# B&R Automation Studio project testovaci_pneu_stan (part 4)

#### multiword_types.h
```c
/*
 * multiword_types.h
 *
 * Academic License - for use in teaching, academic research, and meeting
 * course requirements at degree granting institutions only.  Not for
 * government, commercial, or other organizational use.
 *
 * Code generation for model "reg_FF_PI_pl_regr_stiff".
 *
 * Model version              : 1.135
 * Simulink Coder version : 9.6 (R2021b) 14-May-2021
 * C source code generated on : Tue Sep 27 10:51:43 2022
 *
 * Target selection: bur_grt.tlc
 * Note: GRT includes extra infrastructure and instrumentation for prototyping
 * Embedded hardware selection: Intel->x86/Pentium
 * Code generation objectives: Unspecified
 * Validation result: Not run
 */

#ifndef MULTIWORD_TYPES_H
#define MULTIWORD_TYPES_H
#include "rtwtypes.h"

/*
 * MultiWord supporting definitions
 */
typedef long int long_T;

/*
 * MultiWord types
 */
typedef struct {
  uint32_T chunks[2];
} int64m_T;

typedef struct {
  int64m_T re;
  int64m_T im;
} cint64m_T;

typedef struct {
  uint32_T chunks[2];
} uint64m_T;

typedef struct {
  uint64m_T re;
  uint64m_T im;
} cuint64m_T;

typedef struct {
  uint32_T chunks[3];
} int96m_T;

typedef struct {
  int96m_T re;
  int96m_T im;
} cint96m_T;

typedef struct {
  uint32_T chunks[3];
} uint96m_T;

typedef struct {
  uint96m_T re;
  uint96m_T im;
} cuint96m_T;

typedef struct {
  uint32_T chunks[4];
} int128m_T;

typedef struct {
  int128m_T re;
  int128m_T im;
} cint128m_T;

typedef struct {
  uint32_T chunks[4];
} uint128m_T;

typedef struct {
  uint128m_T re;
  uint128m_T im;
} cuint128m_T;

typedef struct {
  uint32_T chunks[5];
} int160m_T;

typedef struct {
  int160m_T re;
  int160m_T im;
} cint160m_T;

typedef struct {
  uint32_T chunks[5];
} uint160m_T;

typedef struct {
  uint160m_T re;
  uint160m_T im;
} cuint160m_T;

typedef struct {
  uint32_T chunks[6];
} int192m_T;

typedef struct {
  int192m_T re;
  int192m_T im;
} cint192m_T;

typedef struct {
  uint32_T chunks[6];
} uint192m_T;

typedef struct {
  uint192m_T re;
  uint192m_T im;
} cuint192m_T;

typedef struct {
  uint32_T chunks[7];
} int224m_T;

typedef struct {
  int224m_T re;
  int224m_T im;
} cint224m_T;

typedef struct {
  uint32_T chunks[7];
} uint224m_T;

typedef struct {
  uint224m_T re;
  uint224m_T im;
} cuint224m_T;

typedef struct {
  uint32_T chunks[8];
} int256m_T;

typedef struct {
  int256m_T re;
  int256m_T im;
} cint256m_T;

typedef struct {
  uint32_T chunks[8];
} uint256m_T;

typedef struct {
  uint256m_T re;
  uint256m_T im;
} cuint256m_T;

typedef struct {
  uint32_T chunks[9];
} int288m_T;

typedef struct {
  int288m_T re;
  int288m_T im;
} cint288m_T;

typedef struct {
  uint32_T chunks[9];
} uint288m_T;

typedef struct {
  uint288m_T re;
  uint288m_T im;
} cuint288m_T;

typedef struct {
  uint32_T chunks[10];
} int320m_T;

typedef struct {
  int320m_T re;
  int320m_T im;
} cint320m_T;

typedef struct {
  uint32_T chunks[10];
} uint320m_T;

typedef struct {
  uint320m_T re;
  uint320m_T im;
} cuint320m_T;

typedef struct {
  uint32_T chunks[11];
} int352m_T;

typedef struct {
  int352m_T re;
  int352m_T im;
} cint352m_T;

typedef struct {
  uint32_T chunks[11];
} uint352m_T;

typedef struct {
  uint352m_T re;
  uint352m_T im;
} cuint352m_T;

typedef struct {
  uint32_T chunks[12];
} int384m_T;

typedef struct {
  int384m_T re;
  int384m_T im;
} cint384m_T;

typedef struct {
  uint32_T chunks[12];
} uint384m_T;

typedef struct {
  uint384m_T re;
  uint384m_T im;
} cuint384m_T;

typedef struct {
  uint32_T chunks[13];
} int416m_T;

typedef struct {
  int416m_T re;
  int416m_T im;
} cint416m_T;

typedef struct {
  uint32_T chunks[13];
} uint416m_T;

typedef struct {
  uint416m_T re;
  uint416m_T im;
} cuint416m_T;

typedef struct {
  uint32_T chunks[14];
} int448m_T;

typedef struct {
  int448m_T re;
  int448m_T im;
} cint448m_T;

typedef struct {
  uint32_T chunks[14];
} uint448m_T;

typedef struct {
  uint448m_T re;
  uint448m_T im;
} cuint448m_T;

typedef struct {
  uint32_T chunks[15];
} int480m_T;

typedef struct {
  int480m_T re;
  int480m_T im;
} cint480m_T;

typedef struct {
  uint32_T chunks[15];
} uint480m_T;

typedef struct {
  uint480m_T re;
  uint480m_T im;
} cuint480m_T;

typedef struct {
  uint32_T chunks[16];
} int512m_T;

typedef struct {
  int512m_T re;
  int512m_T im;
} cint512m_T;

typedef struct {
  uint32_T chunks[16];
} uint512m_T;

typedef struct {
  uint512m_T re;
  uint512m_T im;
} cuint512m_T;

typedef struct {
  uint32_T chunks[17];
} int544m_T;

typedef struct {
  int544m_T re;
  int544m_T im;
} cint544m_T;

typedef struct {
  uint32_T chunks[17];
} uint544m_T;

typedef struct {
  uint544m_T re;
  uint544m_T im;
} cuint544m_T;

typedef struct {
  uint32_T chunks[18];
} int576m_T;

typedef struct {
  int576m_T re;
  int576m_T im;
} cint576m_T;

typedef struct {
  uint32_T chunks[18];
} uint576m_T;

typedef struct {
  uint576m_T re;
  uint576m_T im;
} cuint576m_T;

typedef struct {
  uint32_T chunks[19];
} int608m_T;

typedef struct {
  int608m_T re;
  int608m_T im;
} cint608m_T;

typedef struct {
  uint32_T chunks[19];
} uint608m_T;

typedef struct {
  uint608m_T re;
  uint608m_T im;
} cuint608m_T;

typedef struct {
  uint32_T chunks[20];
} int640m_T;

typedef struct {
  int640m_T re;
  int640m_T im;
} cint640m_T;

typedef struct {
  uint32_T chunks[20];
} uint640m_T;

typedef struct {
  uint640m_T re;
  uint640m_T im;
} cuint640m_T;

typedef struct {
  uint32_T chunks[21];
} int672m_T;

typedef struct {
  int672m_T re;
  int672m_T im;
} cint672m_T;

typedef struct {
  uint32_T chunks[21];
} uint672m_T;

typedef struct {
  uint672m_T re;
  uint672m_T im;
} cuint672m_T;

typedef struct {
  uint32_T chunks[22];
} int704m_T;

typedef struct {
  int704m_T re;
  int704m_T im;
} cint704m_T;

typedef struct {
  uint32_T chunks[22];
} uint704m_T;

typedef struct {
  uint704m_T re;
  uint704m_T im;
} cuint704m_T;

typedef struct {
  uint32_T chunks[23];
} int736m_T;

typedef struct {
  int736m_T re;
  int736m_T im;
} cint736m_T;

typedef struct {
  uint32_T chunks[23];
} uint736m_T;

typedef struct {
  uint736m_T re;
  uint736m_T im;
} cuint736m_T;

typedef struct {
  uint32_T chunks[24];
} int768m_T;

typedef struct {
  int768m_T re;
  int768m_T im;
} cint768m_T;

typedef struct {
  uint32_T chunks[24];
} uint768m_T;

typedef struct {
  uint768m_T re;
  uint768m_T im;
} cuint768m_T;

typedef struct {
  uint32_T chunks[25];
} int800m_T;

typedef struct {
  int800m_T re;
  int800m_T im;
} cint800m_T;

typedef struct {
  uint32_T chunks[25];
} uint800m_T;

typedef struct {
  uint800m_T re;
  uint800m_T im;
} cuint800m_T;

typedef struct {
  uint32_T chunks[26];
} int832m_T;

typedef struct {
  int832m_T re;
  int832m_T im;
} cint832m_T;

typedef struct {
  uint32_T chunks[26];
} uint832m_T;

typedef struct {
  uint832m_T re;
  uint832m_T im;
} cuint832m_T;

typedef struct {
  uint32_T chunks[27];
} int864m_T;

typedef struct {
  int864m_T re;
  int864m_T im;
} cint864m_T;

typedef struct {
  uint32_T chunks[27];
} uint864m_T;

typedef struct {
  uint864m_T re;
  uint864m_T im;
} cuint864m_T;

typedef struct {
  uint32_T chunks[28];
} int896m_T;

typedef struct {
  int896m_T re;
  int896m_T im;
} cint896m_T;

typedef struct {
  uint32_T chunks[28];
} uint896m_T;

typedef struct {
  uint896m_T re;
  uint896m_T im;
} cuint896m_T;

typedef struct {
  uint32_T chunks[29];
} int928m_T;

typedef struct {
  int928m_T re;
  int928m_T im;
} cint928m_T;

typedef struct {
  uint32_T chunks[29];
} uint928m_T;

typedef struct {
  uint928m_T re;
  uint928m_T im;
} cuint928m_T;

typedef struct {
  uint32_T chunks[30];
} int960m_T;

typedef struct {
  int960m_T re;
  int960m_T im;
} cint960m_T;

typedef struct {
  uint32_T chunks[30];
} uint960m_T;

typedef struct {
  uint960m_T re;
  uint960m_T im;
} cuint960m_T;

typedef struct {
  uint32_T chunks[31];
} int992m_T;

typedef struct {
  int992m_T re;
  int992m_T im;
} cint992m_T;

typedef struct {
  uint32_T chunks[31];
} uint992m_T;

typedef struct {
  uint992m_T re;
  uint992m_T im;
} cuint992m_T;

typedef struct {
  uint32_T chunks[32];
} int1024m_T;

typedef struct {
  int1024m_T re;
  int1024m_T im;
} cint1024m_T;

typedef struct {
  uint32_T chunks[32];
} uint1024m_T;

typedef struct {
  uint1024m_T re;
  uint1024m_T im;
} cuint1024m_T;

typedef struct {
  uint32_T chunks[33];
} int1056m_T;

typedef struct {
  int1056m_T re;
  int1056m_T im;
} cint1056m_T;

typedef struct {
  uint32_T chunks[33];
} uint1056m_T;

typedef struct {
  uint1056m_T re;
  uint1056m_T im;
} cuint1056m_T;

typedef struct {
  uint32_T chunks[34];
} int1088m_T;

typedef struct {
  int1088m_T re;
  int1088m_T im;
} cint1088m_T;

typedef struct {
  uint32_T chunks[34];
} uint1088m_T;

typedef struct {
  uint1088m_T re;
  uint1088m_T im;
} cuint1088m_T;

typedef struct {
  uint32_T chunks[35];
} int1120m_T;

typedef struct {
  int1120m_T re;
  int1120m_T im;
} cint1120m_T;

typedef struct {
  uint32_T chunks[35];
} uint1120m_T;

typedef struct {
  uint1120m_T re;
  uint1120m_T im;
} cuint1120m_T;

typedef struct {
  uint32_T chunks[36];
} int1152m_T;

typedef struct {
  int1152m_T re;
  int1152m_T im;
} cint1152m_T;

typedef struct {
  uint32_T chunks[36];
} uint1152m_T;

typedef struct {
  uint1152m_T re;
  uint1152m_T im;
} cuint1152m_T;

typedef struct {
  uint32_T chunks[37];
} int1184m_T;

typedef struct {
  int1184m_T re;
  int1184m_T im;
} cint1184m_T;

typedef struct {
  uint32_T chunks[37];
} uint1184m_T;

typedef struct {
  uint1184m_T re;
  uint1184m_T im;
} cuint1184m_T;

typedef struct {
  uint32_T chunks[38];
} int1216m_T;

typedef struct {
  int1216m_T re;
  int1216m_T im;
} cint1216m_T;

typedef struct {
  uint32_T chunks[38];
} uint1216m_T;

typedef struct {
  uint1216m_T re;
  uint1216m_T im;
} cuint1216m_T;

typedef struct {
  uint32_T chunks[39];
} int1248m_T;

typedef struct {
  int1248m_T re;
  int1248m_T im;
} cint1248m_T;

typedef struct {
  uint32_T chunks[39];
} uint1248m_T;

typedef struct {
  uint1248m_T re;
  uint1248m_T im;
} cuint1248m_T;

typedef struct {
  uint32_T chunks[40];
} int1280m_T;

typedef struct {
  int1280m_T re;
  int1280m_T im;
} cint1280m_T;

typedef struct {
  uint32_T chunks[40];
} uint1280m_T;

typedef struct {
  uint1280m_T re;
  uint1280m_T im;
} cuint1280m_T;

typedef struct {
  uint32_T chunks[41];
} int1312m_T;

typedef struct {
  int1312m_T re;
  int1312m_T im;
} cint1312m_T;

typedef struct {
  uint32_T chunks[41];
} uint1312m_T;

typedef struct {
  uint1312m_T re;
  uint1312m_T im;
} cuint1312m_T;

typedef struct {
  uint32_T chunks[42];
} int1344m_T;

typedef struct {
  int1344m_T re;
  int1344m_T im;
} cint1344m_T;

typedef struct {
  uint32_T chunks[42];
} uint1344m_T;

typedef struct {
  uint1344m_T re;
  uint1344m_T im;
} cuint1344m_T;

typedef struct {
  uint32_T chunks[43];
} int1376m_T;

typedef struct {
  int1376m_T re;
  int1376m_T im;
} cint1376m_T;

typedef struct {
  uint32_T chunks[43];
} uint1376m_T;

typedef struct {
  uint1376m_T re;
  uint1376m_T im;
} cuint1376m_T;

typedef struct {
  uint32_T chunks[44];
} int1408m_T;

typedef struct {
  int1408m_T re;
  int1408m_T im;
} cint1408m_T;

typedef struct {
  uint32_T chunks[44];
} uint1408m_T;

typedef struct {
  uint1408m_T re;
  uint1408m_T im;
} cuint1408m_T;

typedef struct {
  uint32_T chunks[45];
} int1440m_T;

typedef struct {
  int1440m_T re;
  int1440m_T im;
} cint1440m_T;

typedef struct {
  uint32_T chunks[45];
} uint1440m_T;

typedef struct {
  uint1440m_T re;
  uint1440m_T im;
} cuint1440m_T;

typedef struct {
  uint32_T chunks[46];
} int1472m_T;

typedef struct {
  int1472m_T re;
  int1472m_T im;
} cint1472m_T;

typedef struct {
  uint32_T chunks[46];
} uint1472m_T;

typedef struct {
  uint1472m_T re;
  uint1472m_T im;
} cuint1472m_T;

typedef struct {
  uint32_T chunks[47];
} int1504m_T;

typedef struct {
  int1504m_T re;
  int1504m_T im;
} cint1504m_T;

typedef struct {
  uint32_T chunks[47];
} uint1504m_T;

typedef struct {
  uint1504m_T re;
  uint1504m_T im;
} cuint1504m_T;

typedef struct {
  uint32_T chunks[48];
} int1536m_T;

typedef struct {
  int1536m_T re;
  int1536m_T im;
} cint1536m_T;

typedef struct {
  uint32_T chunks[48];
} uint1536m_T;

typedef struct {
  uint1536m_T re;
  uint1536m_T im;
} cuint1536m_T;

typedef struct {
  uint32_T chunks[49];
} int1568m_T;

typedef struct {
  int1568m_T re;
  int1568m_T im;
} cint1568m_T;

typedef struct {
  uint32_T chunks[49];
} uint1568m_T;

typedef struct {
  uint1568m_T re;
  uint1568m_T im;
} cuint1568m_T;

typedef struct {
  uint32_T chunks[50];
} int1600m_T;

typedef struct {
  int1600m_T re;
  int1600m_T im;
} cint1600m_T;

typedef struct {
  uint32_T chunks[50];
} uint1600m_T;

typedef struct {
  uint1600m_T re;
  uint1600m_T im;
} cuint1600m_T;

typedef struct {
  uint32_T chunks[51];
} int1632m_T;

typedef struct {
  int1632m_T re;
  int1632m_T im;
} cint1632m_T;

typedef struct {
  uint32_T chunks[51];
} uint1632m_T;

typedef struct {
  uint1632m_T re;
  uint1632m_T im;
} cuint1632m_T;

typedef struct {
  uint32_T chunks[52];
} int1664m_T;

typedef struct {
  int1664m_T re;
  int1664m_T im;
} cint1664m_T;

typedef struct {
  uint32_T chunks[52];
} uint1664m_T;

typedef struct {
  uint1664m_T re;
  uint1664m_T im;
} cuint1664m_T;

typedef struct {
  uint32_T chunks[53];
} int1696m_T;

typedef struct {
  int1696m_T re;
  int1696m_T im;
} cint1696m_T;

typedef struct {
  uint32_T chunks[53];
} uint1696m_T;

typedef struct {
  uint1696m_T re;
  uint1696m_T im;
} cuint1696m_T;

typedef struct {
  uint32_T chunks[54];
} int1728m_T;

typedef struct {
  int1728m_T re;
  int1728m_T im;
} cint1728m_T;

typedef struct {
  uint32_T chunks[54];
} uint1728m_T;

typedef struct {
  uint1728m_T re;
  uint1728m_T im;
} cuint1728m_T;

typedef struct {
  uint32_T chunks[55];
} int1760m_T;

typedef struct {
  int1760m_T re;
  int1760m_T im;
} cint1760m_T;

typedef struct {
  uint32_T chunks[55];
} uint1760m_T;

typedef struct {
  uint1760m_T re;
  uint1760m_T im;
} cuint1760m_T;

typedef struct {
  uint32_T chunks[56];
} int1792m_T;

typedef struct {
  int1792m_T re;
  int1792m_T im;
} cint1792m_T;

typedef struct {
  uint32_T chunks[56];
} uint1792m_T;

typedef struct {
  uint1792m_T re;
  uint1792m_T im;
} cuint1792m_T;

typedef struct {
  uint32_T chunks[57];
} int1824m_T;

typedef struct {
  int1824m_T re;
  int1824m_T im;
} cint1824m_T;

typedef struct {
  uint32_T chunks[57];
} uint1824m_T;

typedef struct {
  uint1824m_T re;
  uint1824m_T im;
} cuint1824m_T;

typedef struct {
  uint32_T chunks[58];
} int1856m_T;

typedef struct {
  int1856m_T re;
  int1856m_T im;
} cint1856m_T;

typedef struct {
  uint32_T chunks[58];
} uint1856m_T;

typedef struct {
  uint1856m_T re;
  uint1856m_T im;
} cuint1856m_T;

typedef struct {
  uint32_T chunks[59];
} int1888m_T;

typedef struct {
  int1888m_T re;
  int1888m_T im;
} cint1888m_T;

typedef struct {
  uint32_T chunks[59];
} uint1888m_T;

typedef struct {
  uint1888m_T re;
  uint1888m_T im;
} cuint1888m_T;

typedef struct {
  uint32_T chunks[60];
} int1920m_T;

typedef struct {
  int1920m_T re;
  int1920m_T im;
} cint1920m_T;

typedef struct {
  uint32_T chunks[60];
} uint1920m_T;

typedef struct {
  uint1920m_T re;
  uint1920m_T im;
} cuint1920m_T;

typedef struct {
  uint32_T chunks[61];
} int1952m_T;

typedef struct {
  int1952m_T re;
  int1952m_T im;
} cint1952m_T;

typedef struct {
  uint32_T chunks[61];
} uint1952m_T;

typedef struct {
  uint1952m_T re;
  uint1952m_T im;
} cuint1952m_T;

typedef struct {
  uint32_T chunks[62];
} int1984m_T;

typedef struct {
  int1984m_T re;
  int1984m_T im;
} cint1984m_T;

typedef struct {
  uint32_T chunks[62];
} uint1984m_T;

typedef struct {
  uint1984m_T re;
  uint1984m_T im;
} cuint1984m_T;

typedef struct {
  uint32_T chunks[63];
} int2016m_T;

typedef struct {
  int2016m_T re;
  int2016m_T im;
} cint2016m_T;

typedef struct {
  uint32_T chunks[63];
} uint2016m_T;

typedef struct {
  uint2016m_T re;
  uint2016m_T im;
} cuint2016m_T;

typedef struct {
  uint32_T chunks[64];
} int2048m_T;

typedef struct {
  int2048m_T re;
  int2048m_T im;
} cint2048m_T;

typedef struct {
  uint32_T chunks[64];
} uint2048m_T;

typedef struct {
  uint2048m_T re;
  uint2048m_T im;
} cuint2048m_T;

#endif                                 /* MULTIWORD_TYPES_H */
```

#### rtwtypes.h
```c
/*
 * rtwtypes.h
 *
 * Academic License - for use in teaching, academic research, and meeting
 * course requirements at degree granting institutions only.  Not for
 * government, commercial, or other organizational use.
 *
 * Code generation for model "reg_FF_PI_pl_regr_stiff".
 *
 * Model version              : 1.135
 * Simulink Coder version : 9.6 (R2021b) 14-May-2021
 * C source code generated on : Tue Sep 27 10:51:43 2022
 *
 * Target selection: bur_grt.tlc
 * Note: GRT includes extra infrastructure and instrumentation for prototyping
 * Embedded hardware selection: Intel->x86/Pentium
 * Code generation objectives: Unspecified
 * Validation result: Not run
 */

#ifndef RTWTYPES_H
#define RTWTYPES_H
#include "tmwtypes.h"
#ifndef POINTER_T
#define POINTER_T

typedef void * pointer_T;

#endif

/* Logical type definitions */
#if (!defined(__cplusplus))
#ifndef false
#define false                          (0U)
#endif

#ifndef true
#define true                           (1U)
#endif
#endif
#endif                                 /* RTWTYPES_H */
```

#### FF_PID_r_t.c
```c
/********************************************************************
 * COPYRIGHT -- B&R Industrial Automation GmbH
 ********************************************************************
 * Program: regulatory
 * File: regulatory.c
 * Author: MartinV
 * Last modified by: MartinV
 * Created: 27-Sep-2022 10:51:51
 * Last modified: Tue Sep 27 10:50:57 2022
 * Model Version: 1.135
 * Description:
 * modified Comment:
 ********************************************************************
 * Implementation of program regulatory
 ********************************************************************
 * Generated with B&R Automation Studio Target for Simulink V6.5
 * (GRT based)
 ********************************************************************/

#include <bur/plctypes.h>

#include "rtwtypes.h"
#include "rtmodel.h"

#define EXPAND_CONCAT(name1,name2) name1 ## name2
#define CONCAT(name1,name2) EXPAND_CONCAT(name1,name2)
#define RT_MODEL            CONCAT(MODEL,_rtModel)

#ifdef __cplusplus

extern "C" {

#endif

/* Defines */
#define SS_TERMINATE 4
#define SS_OUTPUT 3
#define SS_INITIALIZE 2

#ifdef __cplusplus

}

#endif

#ifdef __cplusplus
    unsigned long bur_heap_size = 6553500;
#endif

void FF_PID_r_t(struct FF_PID_r_t* inst)
{
  tag_RTM_reg_FF_PI_pl_regr_sti_T* const reg_FF_PI_pl_regr_stiff_M = &(inst)->bur_reg_FF_PI_pl_regr_stiff;
	inst->bur_reg_FF_PI_pl_regr_stiff.blockIO = &(inst)->bur_B_reg_FF_PI_pl_regr_stiff_T;
	inst->bur_reg_FF_PI_pl_regr_stiff.dwork = &(inst)->bur_DW_reg_FF_PI_pl_regr_stiff_;

  switch (inst->ssMethodType)
  {
    case SS_INITIALIZE:

      /* call model initialize functions */
		/*memInit function */
		reg_FF_PI_pl_regr_stiff_initializeMemory(reg_FF_PI_pl_regr_stiff_M, inst);
		reg_FF_PI_pl_regr_stiff_initialize(reg_FF_PI_pl_regr_stiff_M, inst);
      break;

    case SS_OUTPUT:
      /* call model step functions */
		reg_FF_PI_pl_regr_stiff_step(reg_FF_PI_pl_regr_stiff_M, inst);
      break;

    case SS_TERMINATE:
      /* call model terminate function */
		reg_FF_PI_pl_regr_stiff_terminate(reg_FF_PI_pl_regr_stiff_M, inst);
	  break;
  }
}

/*****************************************************************************
   Function block sample time: 0.002
 *****************************************************************************/

/*****************************************************************************
   B&R Automation Studio Target for Simulink Version: V6.5.1 (03-Dec-2021)
 *****************************************************************************/
```

#### reg_FF_PI_pl_regr_stiff.c
```c
/*
 * reg_FF_PI_pl_regr_stiff.c
 *
 * Academic License - for use in teaching, academic research, and meeting
 * course requirements at degree granting institutions only.  Not for
 * government, commercial, or other organizational use.
 *
 * Code generation for model "reg_FF_PI_pl_regr_stiff".
 *
 * Model version              : 1.135
 * Simulink Coder version : 9.6 (R2021b) 14-May-2021
 * C source code generated on : Tue Sep 27 10:51:43 2022
 *
 * Target selection: bur_grt.tlc
 * Note: GRT includes extra infrastructure and instrumentation for prototyping
 * Embedded hardware selection: Intel->x86/Pentium
 * Code generation objectives: Unspecified
 * Validation result: Not run
 */

#include "reg_FF_PI_pl_regr_stiff.h"
#include "reg_FF_PI_pl_regr_stiff_private.h"

/* Forward declaration for local functions */
static real32_T reg_FF_PI_pl_regr_stiff_norm(const real32_T x[4], struct FF_PID_r_t* inst);

/* Function for MATLAB Function: '<S4>/requested alfa 2 deltaz1' */
static real32_T reg_FF_PI_pl_regr_stiff_norm(const real32_T x[4], struct FF_PID_r_t* inst)
{
  real32_T absxk;
  real32_T scale;
  real32_T t;
  real32_T y;
  scale = 1.29246971E-26F;
  absxk = fabsf(x[0]);
  if (absxk > 1.29246971E-26F) {
    y = 1.0F;
    scale = absxk;
  } else {
    t = absxk / 1.29246971E-26F;
    y = t * t;
  }

  absxk = fabsf(x[1]);
  if (absxk > scale) {
    t = scale / absxk;
    y = y * t * t + 1.0F;
    scale = absxk;
  } else {
    t = absxk / scale;
    y += t * t;
  }

  absxk = fabsf(x[2]);
  if (absxk > scale) {
    t = scale / absxk;
    y = y * t * t + 1.0F;
    scale = absxk;
  } else {
    t = absxk / scale;
    y += t * t;
  }

  absxk = fabsf(x[3]);
  if (absxk > scale) {
    t = scale / absxk;
    y = y * t * t + 1.0F;
    scale = absxk;
  } else {
    t = absxk / scale;
    y += t * t;
  }

  return scale * sqrtf(y);
}

/* Model step function */
void reg_FF_PI_pl_regr_stiff_step(RT_MODEL_reg_FF_PI_pl_regr_st_T *const
  reg_FF_PI_pl_regr_stiff_M, struct FF_PID_r_t* inst)
{
  B_reg_FF_PI_pl_regr_stiff_T *reg_FF_PI_pl_regr_stiff_B =
    reg_FF_PI_pl_regr_stiff_M->blockIO;
  DW_reg_FF_PI_pl_regr_stiff_T *reg_FF_PI_pl_regr_stiff_DW =
    reg_FF_PI_pl_regr_stiff_M->dwork;
  real_T Tz23[16];
  real_T Blue0_tmp[4];
  real_T Yellow0_tmp[4];
  real_T A1;
  real_T A2;
  real_T A3;
  real_T rtb_Sum1;
  real_T rtb_Sum2;
  real_T rtb_Sum_d;
  real_T rtb_Switch1;
  int32_T Tz23_tmp;
  int32_T Tz23_tmp_tmp;
  int32_T i;
  int32_T i_0;
  real32_T AlphaY_0[16];
  real32_T HTransform[16];
  real32_T HTransform_tmp_3[16];
  real32_T Tz23_0[16];
  real32_T tmp[8];
  real32_T tmp_0[6];
  real32_T tmp_1[6];
  real32_T Blue0_tmp_0[4];
  real32_T Green0_tmp_tmp_0[4];
  real32_T Yellow0_tmp_0[4];
  real32_T Yellow0_tmp_1[4];
  real32_T AlphaX;
  real32_T AlphaY;
  real32_T HTransform_tmp;
  real32_T HTransform_tmp_0;
  real32_T tmp_2;
  real32_T tmp_3;
  real32_T tmp_4;
  real32_T tmp_5;
  real32_T tmp_6;
  real32_T tmp_7;
  real32_T tmp_8;
  real32_T tmp_9;
  real32_T tmp_a;
  real32_T tmp_b;
  real32_T tmp_c;
  int8_T Green0_tmp_tmp[4];
  int8_T HTransform_tmp_1[4];
  int8_T HTransform_tmp_2[4];

  /* S-Function (bur_in): '<Root>/Input15' */
  reg_FF_PI_pl_regr_stiff_B->Input15 = inst->stiffness_ff;

  /* S-Function (bur_in): '<Root>/Input1' */
  reg_FF_PI_pl_regr_stiff_B->Input1 = inst->ref_alfa_x;

  /* S-Function (bur_in): '<Root>/Input2' */
  reg_FF_PI_pl_regr_stiff_B->Input2 = inst->ref_alfa_y;

  /* S-Function (bur_in): '<Root>/Input3' */
  reg_FF_PI_pl_regr_stiff_B->Input3 = inst->real_alfa_x;

  /* S-Function (bur_in): '<Root>/Input4' */
  reg_FF_PI_pl_regr_stiff_B->Input4 = inst->real_alfa_y;

  /* MATLAB Function: '<S4>/requested alfa 2 deltaz1' incorporates:
   *  Constant: '<S4>/Constant1'
   */
  AlphaX = reg_FF_PI_pl_regr_stiff_B->Input1 * 3.14159274F / 180.0F;
  AlphaY = -reg_FF_PI_pl_regr_stiff_B->Input2 * 3.14159274F / 180.0F;
  Tz23[2] = 0.0;
  Tz23[6] = 0.0;
  Tz23[10] = 1.0;
  Tz23[14] = 57.5;
  HTransform_tmp = sinf(AlphaY);
  AlphaY = cosf(AlphaY);
  HTransform_tmp_0 = sinf(AlphaX);
  AlphaX = cosf(AlphaX);
  AlphaY_0[0] = AlphaY;
  AlphaY_0[4] = 0.0F;
  AlphaY_0[8] = HTransform_tmp;
  AlphaY_0[12] = 0.0F;
  AlphaY_0[2] = -HTransform_tmp;
  AlphaY_0[6] = 0.0F;
  AlphaY_0[10] = AlphaY;
  AlphaY_0[14] = 0.0F;
  Tz23[0] = 1.0;
  Tz23[1] = 0.0;
  Tz23[3] = 0.0;
  HTransform_tmp_2[0] = 1;
  AlphaY_0[1] = 0.0F;
  AlphaY_0[3] = 0.0F;
  HTransform_tmp_1[0] = 0;
  Tz23[4] = 0.0;
  Tz23[5] = 1.0;
  Tz23[7] = 0.0;
  HTransform_tmp_2[1] = 0;
  AlphaY_0[5] = 1.0F;
  AlphaY_0[7] = 0.0F;
  HTransform_tmp_1[1] = 0;
  Tz23[8] = 0.0;
  Tz23[9] = 0.0;
  Tz23[11] = 0.0;
  HTransform_tmp_2[2] = 0;
  AlphaY_0[9] = 0.0F;
  AlphaY_0[11] = 0.0F;
  HTransform_tmp_1[2] = 0;
  Tz23[12] = 0.0;
  Tz23[13] = 0.0;
  Tz23[15] = 1.0;
  HTransform_tmp_2[3] = 0;
  AlphaY_0[13] = 0.0F;
  AlphaY_0[15] = 1.0F;
  HTransform_tmp_1[3] = 1;
  HTransform_tmp_3[1] = 0.0F;
  HTransform_tmp_3[5] = AlphaX;
  HTransform_tmp_3[9] = -HTransform_tmp_0;
  HTransform_tmp_3[13] = 0.0F;
  HTransform_tmp_3[2] = 0.0F;
  HTransform_tmp_3[6] = HTransform_tmp_0;
  HTransform_tmp_3[10] = AlphaX;
  HTransform_tmp_3[14] = 0.0F;
  for (i = 0; i < 4; i++) {
    for (i_0 = 0; i_0 < 4; i_0++) {
      Tz23_tmp_tmp = i_0 << 2;
      Tz23_tmp = i + Tz23_tmp_tmp;
      Tz23_0[Tz23_tmp] = 0.0F;
      Tz23_0[Tz23_tmp] += AlphaY_0[Tz23_tmp_tmp] * (real32_T)Tz23[i];
      Tz23_0[Tz23_tmp] += AlphaY_0[Tz23_tmp_tmp + 1] * (real32_T)Tz23[i + 4];
      Tz23_0[Tz23_tmp] += AlphaY_0[Tz23_tmp_tmp + 2] * (real32_T)Tz23[i + 8];
      Tz23_0[Tz23_tmp] += AlphaY_0[Tz23_tmp_tmp + 3] * (real32_T)Tz23[i + 12];
    }

    Tz23_tmp_tmp = i << 2;
    HTransform_tmp_3[Tz23_tmp_tmp] = HTransform_tmp_2[i];
    HTransform_tmp_3[Tz23_tmp_tmp + 3] = HTransform_tmp_1[i];
  }

  Green0_tmp_tmp[0] = 85;
  Green0_tmp_tmp[1] = 0;
  Green0_tmp_tmp[2] = 0;
  Green0_tmp_tmp[3] = 1;
  Yellow0_tmp[0] = -42.5;
  Yellow0_tmp[1] = 73.612159321677282;
  Yellow0_tmp[2] = 0.0;
  Yellow0_tmp[3] = 1.0;
  Blue0_tmp[0] = -42.5;
  Blue0_tmp[1] = -73.612159321677282;
  Blue0_tmp[2] = 0.0;
  Blue0_tmp[3] = 1.0;
  for (i = 0; i < 4; i++) {
    for (i_0 = 0; i_0 < 4; i_0++) {
      Tz23_tmp_tmp = i_0 << 2;
      Tz23_tmp = i + Tz23_tmp_tmp;
      AlphaY_0[Tz23_tmp] = 0.0F;
      AlphaY_0[Tz23_tmp] += HTransform_tmp_3[Tz23_tmp_tmp] * Tz23_0[i];
      AlphaY_0[Tz23_tmp] += HTransform_tmp_3[Tz23_tmp_tmp + 1] * Tz23_0[i + 4];
      AlphaY_0[Tz23_tmp] += HTransform_tmp_3[Tz23_tmp_tmp + 2] * Tz23_0[i + 8];
      AlphaY_0[Tz23_tmp] += HTransform_tmp_3[Tz23_tmp_tmp + 3] * Tz23_0[i + 12];
    }

    AlphaX = 0.0F;
    AlphaY = 0.0F;
    HTransform_tmp = 0.0F;
    for (i_0 = 0; i_0 < 4; i_0++) {
      Tz23_tmp_tmp = i_0 << 2;
      Tz23_tmp = i + Tz23_tmp_tmp;
      HTransform[Tz23_tmp] = 0.0F;
      HTransform[Tz23_tmp] += (real32_T)Tz23[Tz23_tmp_tmp] * AlphaY_0[i];
      HTransform[Tz23_tmp] += (real32_T)Tz23[Tz23_tmp_tmp + 1] * AlphaY_0[i + 4];
      HTransform[Tz23_tmp] += (real32_T)Tz23[Tz23_tmp_tmp + 2] * AlphaY_0[i + 8];
      HTransform[Tz23_tmp] += (real32_T)Tz23[Tz23_tmp_tmp + 3] * AlphaY_0[i + 12];
      AlphaX += HTransform[Tz23_tmp] * (real32_T)Green0_tmp_tmp[i_0];
      AlphaY += HTransform[Tz23_tmp] * (real32_T)Yellow0_tmp[i_0];
      HTransform_tmp += HTransform[Tz23_tmp] * (real32_T)Blue0_tmp[i_0];
    }

    Green0_tmp_tmp_0[i] = (real32_T)Green0_tmp_tmp[i] - AlphaX;
    Yellow0_tmp_0[i] = (real32_T)Yellow0_tmp[i] - AlphaY;
    Blue0_tmp_0[i] = (real32_T)Blue0_tmp[i] - HTransform_tmp;
  }

  AlphaX = reg_FF_PI_pl_regr_stiff_B->Input3 * 3.14159274F / 180.0F;
  AlphaY = -reg_FF_PI_pl_regr_stiff_B->Input4 * 3.14159274F / 180.0F;
  HTransform_tmp = sinf(AlphaY);
  AlphaY = cosf(AlphaY);
  HTransform_tmp_0 = sinf(AlphaX);
  AlphaX = cosf(AlphaX);
  AlphaY_0[0] = AlphaY;
  AlphaY_0[4] = 0.0F;
  AlphaY_0[8] = HTransform_tmp;
  AlphaY_0[12] = 0.0F;
  AlphaY_0[2] = -HTransform_tmp;
  AlphaY_0[6] = 0.0F;
  AlphaY_0[10] = AlphaY;
  AlphaY_0[14] = 0.0F;
  AlphaY_0[1] = 0.0F;
  AlphaY_0[3] = 0.0F;
  AlphaY_0[5] = 1.0F;
  AlphaY_0[7] = 0.0F;
  AlphaY_0[9] = 0.0F;
  AlphaY_0[11] = 0.0F;
  AlphaY_0[13] = 0.0F;
  AlphaY_0[15] = 1.0F;
  HTransform_tmp_3[1] = 0.0F;
  HTransform_tmp_3[5] = AlphaX;
  HTransform_tmp_3[9] = -HTransform_tmp_0;
  HTransform_tmp_3[13] = 0.0F;
  HTransform_tmp_3[2] = 0.0F;
  HTransform_tmp_3[6] = HTransform_tmp_0;
  HTransform_tmp_3[10] = AlphaX;
  HTransform_tmp_3[14] = 0.0F;
  for (i = 0; i < 4; i++) {
    for (i_0 = 0; i_0 < 4; i_0++) {
      Tz23_tmp_tmp = i_0 << 2;
      Tz23_tmp = i + Tz23_tmp_tmp;
      Tz23_0[Tz23_tmp] = 0.0F;
      Tz23_0[Tz23_tmp] += AlphaY_0[Tz23_tmp_tmp] * (real32_T)Tz23[i];
      Tz23_0[Tz23_tmp] += AlphaY_0[Tz23_tmp_tmp + 1] * (real32_T)Tz23[i + 4];
      Tz23_0[Tz23_tmp] += AlphaY_0[Tz23_tmp_tmp + 2] * (real32_T)Tz23[i + 8];
      Tz23_0[Tz23_tmp] += AlphaY_0[Tz23_tmp_tmp + 3] * (real32_T)Tz23[i + 12];
    }

    Tz23_tmp_tmp = i << 2;
    HTransform_tmp_3[Tz23_tmp_tmp] = HTransform_tmp_2[i];
    HTransform_tmp_3[Tz23_tmp_tmp + 3] = HTransform_tmp_1[i];
  }

  Yellow0_tmp[0] = -42.5;
  Yellow0_tmp[1] = 73.612159321677282;
  Yellow0_tmp[2] = 0.0;
  Yellow0_tmp[3] = 1.0;
  Blue0_tmp[0] = -42.5;
  Blue0_tmp[1] = -73.612159321677282;
  Blue0_tmp[2] = 0.0;
  Blue0_tmp[3] = 1.0;
  for (i = 0; i < 4; i++) {
    for (i_0 = 0; i_0 < 4; i_0++) {
      Tz23_tmp_tmp = i_0 << 2;
      Tz23_tmp = i + Tz23_tmp_tmp;
      AlphaY_0[Tz23_tmp] = 0.0F;
      AlphaY_0[Tz23_tmp] += HTransform_tmp_3[Tz23_tmp_tmp] * Tz23_0[i];
      AlphaY_0[Tz23_tmp] += HTransform_tmp_3[Tz23_tmp_tmp + 1] * Tz23_0[i + 4];
      AlphaY_0[Tz23_tmp] += HTransform_tmp_3[Tz23_tmp_tmp + 2] * Tz23_0[i + 8];
      AlphaY_0[Tz23_tmp] += HTransform_tmp_3[Tz23_tmp_tmp + 3] * Tz23_0[i + 12];
    }

    AlphaX = 0.0F;
    for (i_0 = 0; i_0 < 4; i_0++) {
      Tz23_tmp_tmp = i_0 << 2;
      Tz23_tmp = i + Tz23_tmp_tmp;
      HTransform[Tz23_tmp] = 0.0F;
      HTransform[Tz23_tmp] += (real32_T)Tz23[Tz23_tmp_tmp] * AlphaY_0[i];
      HTransform[Tz23_tmp] += (real32_T)Tz23[Tz23_tmp_tmp + 1] * AlphaY_0[i + 4];
      HTransform[Tz23_tmp] += (real32_T)Tz23[Tz23_tmp_tmp + 2] * AlphaY_0[i + 8];
      HTransform[Tz23_tmp] += (real32_T)Tz23[Tz23_tmp_tmp + 3] * AlphaY_0[i + 12];
      AlphaX += HTransform[Tz23_tmp] * (real32_T)Yellow0_tmp[i_0];
    }

    Yellow0_tmp_1[i] = (real32_T)Yellow0_tmp[i] - AlphaX;
  }

  /* Sum: '<S2>/Sum' incorporates:
   *  Constant: '<S10>/cylinder height'
   *  Constant: '<S8>/cylinder height'
   *  Gain: '<S4>/Gain'
   *  Gain: '<S4>/Gain3'
   *  MATLAB Function: '<S4>/requested alfa 2 deltaz1'
   *  Sum: '<S10>/Sum'
   *  Sum: '<S8>/Sum'
   */
  A2 = (0.001F * reg_FF_PI_pl_regr_stiff_norm(Yellow0_tmp_1, inst) - 0.115) - (0.001F *
    reg_FF_PI_pl_regr_stiff_norm(Yellow0_tmp_0, inst) - 0.115);

  /* S-Function (bur_in): '<Root>/Input11' */
  reg_FF_PI_pl_regr_stiff_B->Input11 = inst->P_parameter;

  /* S-Function (bur_in): '<Root>/Input5' */
  reg_FF_PI_pl_regr_stiff_B->Input5 = inst->reset_PID_blue;

  /* DiscreteIntegrator: '<S144>/Integrator' */
  if ((reg_FF_PI_pl_regr_stiff_B->Input5 <= 0.0F) &&
      (reg_FF_PI_pl_regr_stiff_DW->Integrator_PrevResetState == 1)) {
    reg_FF_PI_pl_regr_stiff_DW->Integrator_DSTATE = 0.0;
  }

  /* S-Function (bur_in): '<Root>/Input13' */
  reg_FF_PI_pl_regr_stiff_B->Input13 = inst->D_parameter;

  /* DiscreteIntegrator: '<S139>/Filter' */
  if ((reg_FF_PI_pl_regr_stiff_B->Input5 <= 0.0F) &&
      (reg_FF_PI_pl_regr_stiff_DW->Filter_PrevResetState == 1)) {
    reg_FF_PI_pl_regr_stiff_DW->Filter_DSTATE = 0.0;
  }

  /* S-Function (bur_in): '<Root>/Input14' */
  reg_FF_PI_pl_regr_stiff_B->Input14 = inst->N_parameter;

  /* Product: '<S147>/NProd Out' incorporates:
   *  DiscreteIntegrator: '<S139>/Filter'
   *  Product: '<S138>/DProd Out'
   *  Sum: '<S139>/SumD'
   */
  A1 = (A2 * reg_FF_PI_pl_regr_stiff_B->Input13 -
        reg_FF_PI_pl_regr_stiff_DW->Filter_DSTATE) *
    reg_FF_PI_pl_regr_stiff_B->Input14;

  /* Switch: '<Root>/Switch2' */
  if (reg_FF_PI_pl_regr_stiff_B->Input5 > 0.0F) {
    /* Sum: '<S154>/Sum' incorporates:
     *  DiscreteIntegrator: '<S144>/Integrator'
     *  Product: '<S149>/PProd Out'
     */
    A3 = (A2 * reg_FF_PI_pl_regr_stiff_B->Input11 +
          reg_FF_PI_pl_regr_stiff_DW->Integrator_DSTATE) + A1;

    /* Switch: '<S152>/Switch2' incorporates:
     *  Constant: '<S2>/max_sat'
     *  Constant: '<S2>/min_sat'
     *  RelationalOperator: '<S152>/LowerRelop1'
     *  RelationalOperator: '<S152>/UpperRelop'
     *  Sum: '<S2>/Sum3'
     *  Sum: '<S2>/Sum4'
     *  Switch: '<S152>/Switch'
     */
    if (A3 > 5.0 - reg_FF_PI_pl_regr_stiff_B->Input15) {
      rtb_Switch1 = 5.0 - reg_FF_PI_pl_regr_stiff_B->Input15;
    } else if (A3 < 0.0 - reg_FF_PI_pl_regr_stiff_B->Input15) {
      /* Switch: '<S152>/Switch' incorporates:
       *  Constant: '<S2>/min_sat'
       *  Sum: '<S2>/Sum4'
       */
      rtb_Switch1 = 0.0 - reg_FF_PI_pl_regr_stiff_B->Input15;
    } else {
      rtb_Switch1 = A3;
    }

    /* End of Switch: '<S152>/Switch2' */
  } else {
    rtb_Switch1 = 0.0;
  }

  /* End of Switch: '<Root>/Switch2' */

  /* MATLAB Function: '<S1>/MATLAB Function' incorporates:
   *  Constant: '<S1>/Constant'
   */
  AlphaX = powf(reg_FF_PI_pl_regr_stiff_B->Input15, 7.0F);
  tmp[0] = AlphaX;
  AlphaY = powf(reg_FF_PI_pl_regr_stiff_B->Input15, 6.0F);
  tmp[1] = AlphaY;
  HTransform_tmp = powf(reg_FF_PI_pl_regr_stiff_B->Input15, 5.0F);
  tmp[2] = HTransform_tmp;
  HTransform_tmp_0 = powf(reg_FF_PI_pl_regr_stiff_B->Input15, 4.0F);
  tmp[3] = HTransform_tmp_0;
  tmp_b = powf(reg_FF_PI_pl_regr_stiff_B->Input15, 3.0F);
  tmp[4] = tmp_b;
  tmp_c = reg_FF_PI_pl_regr_stiff_B->Input15 *
    reg_FF_PI_pl_regr_stiff_B->Input15;
  tmp[5] = tmp_c;
  tmp[6] = reg_FF_PI_pl_regr_stiff_B->Input15;
  tmp[7] = 1.0F;
  tmp_2 = 0.0F;
  for (i = 0; i < 8; i++) {
    tmp_2 += (real32_T)reg_FF_PI_pl_regr_stiff_ConstP.Constant_Value[6 * i] *
      tmp[i];
  }

  tmp[0] = AlphaX;
  tmp[1] = AlphaY;
  tmp[2] = HTransform_tmp;
  tmp[3] = HTransform_tmp_0;
  tmp[4] = tmp_b;
  tmp[5] = tmp_c;
  tmp[6] = reg_FF_PI_pl_regr_stiff_B->Input15;
  tmp[7] = 1.0F;
  tmp_3 = 0.0F;
  for (i = 0; i < 8; i++) {
    tmp_3 += (real32_T)reg_FF_PI_pl_regr_stiff_ConstP.Constant_Value[6 * i + 1] *
      tmp[i];
  }

  tmp[0] = AlphaX;
  tmp[1] = AlphaY;
  tmp[2] = HTransform_tmp;
  tmp[3] = HTransform_tmp_0;
  tmp[4] = tmp_b;
  tmp[5] = tmp_c;
  tmp[6] = reg_FF_PI_pl_regr_stiff_B->Input15;
  tmp[7] = 1.0F;
  tmp_4 = 0.0F;
  for (i = 0; i < 8; i++) {
    tmp_4 += (real32_T)reg_FF_PI_pl_regr_stiff_ConstP.Constant_Value[6 * i + 2] *
      tmp[i];
  }

  tmp[0] = AlphaX;
  tmp[1] = AlphaY;
  tmp[2] = HTransform_tmp;
  tmp[3] = HTransform_tmp_0;
  tmp[4] = tmp_b;
  tmp[5] = tmp_c;
  tmp[6] = reg_FF_PI_pl_regr_stiff_B->Input15;
  tmp[7] = 1.0F;
  tmp_5 = 0.0F;
  for (i = 0; i < 8; i++) {
    tmp_5 += (real32_T)reg_FF_PI_pl_regr_stiff_ConstP.Constant_Value[6 * i + 3] *
      tmp[i];
  }

  tmp[0] = AlphaX;
  tmp[1] = AlphaY;
  tmp[2] = HTransform_tmp;
  tmp[3] = HTransform_tmp_0;
  tmp[4] = tmp_b;
  tmp[5] = tmp_c;
  tmp[6] = reg_FF_PI_pl_regr_stiff_B->Input15;
  tmp[7] = 1.0F;
  tmp_6 = 0.0F;
  for (i = 0; i < 8; i++) {
    tmp_6 += (real32_T)reg_FF_PI_pl_regr_stiff_ConstP.Constant_Value[6 * i + 4] *
      tmp[i];
  }

  tmp[0] = AlphaX;
  tmp[1] = AlphaY;
  tmp[2] = HTransform_tmp;
  tmp[3] = HTransform_tmp_0;
  tmp[4] = tmp_b;
  tmp[5] = tmp_c;
  tmp[6] = reg_FF_PI_pl_regr_stiff_B->Input15;
  tmp[7] = 1.0F;
  tmp_7 = 0.0F;
  for (i = 0; i < 8; i++) {
    tmp_7 += (real32_T)reg_FF_PI_pl_regr_stiff_ConstP.Constant_Value[6 * i + 5] *
      tmp[i];
  }

  tmp_0[0] = tmp_2;
  tmp_0[1] = tmp_3;
  tmp_0[2] = tmp_4;
  tmp_0[3] = tmp_5;
  tmp_0[4] = tmp_6;
  tmp_0[5] = tmp_7;
  tmp_1[0] = 1.0F;
  tmp_1[1] = reg_FF_PI_pl_regr_stiff_B->Input1;
  tmp_1[2] = reg_FF_PI_pl_regr_stiff_B->Input2;
  tmp_2 = reg_FF_PI_pl_regr_stiff_B->Input1 * reg_FF_PI_pl_regr_stiff_B->Input1;
  tmp_1[3] = tmp_2;
  tmp_3 = reg_FF_PI_pl_regr_stiff_B->Input1 * reg_FF_PI_pl_regr_stiff_B->Input2;
  tmp_1[4] = tmp_3;
  tmp_4 = reg_FF_PI_pl_regr_stiff_B->Input2 * reg_FF_PI_pl_regr_stiff_B->Input2;
  tmp_1[5] = tmp_4;
  tmp_5 = 0.0F;
  for (i = 0; i < 6; i++) {
    tmp_5 += tmp_0[i] * tmp_1[i];
  }

  /* Sum: '<Root>/Sum' incorporates:
   *  MATLAB Function: '<S1>/MATLAB Function'
   */
  reg_FF_PI_pl_regr_stiff_B->Sum = (real32_T)(rtb_Switch1 + tmp_5);

  /* S-Function (bur_out): '<Root>/Output1' */
  inst->Blue_tab = reg_FF_PI_pl_regr_stiff_B->Sum;

  /* MATLAB Function: '<S4>/requested alfa 2 deltaz1' */
  for (i = 0; i < 4; i++) {
    Yellow0_tmp_0[i] = (real32_T)Green0_tmp_tmp[i] - (HTransform[i] * 85.0F +
      HTransform[i + 12]);
  }

  /* Sum: '<S2>/Sum2' incorporates:
   *  Constant: '<S11>/cylinder height'
   *  Constant: '<S13>/cylinder height'
   *  Gain: '<S4>/Gain1'
   *  Gain: '<S4>/Gain4'
   *  MATLAB Function: '<S4>/requested alfa 2 deltaz1'
   *  Sum: '<S11>/Sum'
   *  Sum: '<S13>/Sum'
   */
  rtb_Sum2 = (0.001F * reg_FF_PI_pl_regr_stiff_norm(Yellow0_tmp_0, inst) - 0.115) -
    (0.001F * reg_FF_PI_pl_regr_stiff_norm(Green0_tmp_tmp_0, inst) - 0.115);

  /* S-Function (bur_in): '<Root>/Input7' */
  reg_FF_PI_pl_regr_stiff_B->Input7 = inst->reset_PID_green;

  /* DiscreteIntegrator: '<S95>/Integrator' */
  if ((reg_FF_PI_pl_regr_stiff_B->Input7 <= 0.0F) &&
      (reg_FF_PI_pl_regr_stiff_DW->Integrator_PrevResetState_l == 1)) {
    reg_FF_PI_pl_regr_stiff_DW->Integrator_DSTATE_o = 0.0;
  }

  /* DiscreteIntegrator: '<S90>/Filter' */
  if ((reg_FF_PI_pl_regr_stiff_B->Input7 <= 0.0F) &&
      (reg_FF_PI_pl_regr_stiff_DW->Filter_PrevResetState_e == 1)) {
    reg_FF_PI_pl_regr_stiff_DW->Filter_DSTATE_f = 0.0;
  }

  /* Product: '<S98>/NProd Out' incorporates:
   *  DiscreteIntegrator: '<S90>/Filter'
   *  Product: '<S89>/DProd Out'
   *  Sum: '<S90>/SumD'
   */
  A3 = (rtb_Sum2 * reg_FF_PI_pl_regr_stiff_B->Input13 -
        reg_FF_PI_pl_regr_stiff_DW->Filter_DSTATE_f) *
    reg_FF_PI_pl_regr_stiff_B->Input14;

  /* Switch: '<Root>/Switch' */
  if (reg_FF_PI_pl_regr_stiff_B->Input7 > 0.0F) {
    /* Sum: '<S105>/Sum' incorporates:
     *  DiscreteIntegrator: '<S95>/Integrator'
     *  Product: '<S100>/PProd Out'
     */
    rtb_Sum_d = (rtb_Sum2 * reg_FF_PI_pl_regr_stiff_B->Input11 +
                 reg_FF_PI_pl_regr_stiff_DW->Integrator_DSTATE_o) + A3;

    /* Switch: '<S103>/Switch2' incorporates:
     *  Constant: '<S2>/max_sat'
     *  Constant: '<S2>/min_sat'
     *  RelationalOperator: '<S103>/LowerRelop1'
     *  RelationalOperator: '<S103>/UpperRelop'
     *  Sum: '<S2>/Sum3'
     *  Sum: '<S2>/Sum4'
     *  Switch: '<S103>/Switch'
     */
    if (rtb_Sum_d > 5.0 - reg_FF_PI_pl_regr_stiff_B->Input15) {
      rtb_Switch1 = 5.0 - reg_FF_PI_pl_regr_stiff_B->Input15;
    } else if (rtb_Sum_d < 0.0 - reg_FF_PI_pl_regr_stiff_B->Input15) {
      /* Switch: '<S103>/Switch' incorporates:
       *  Constant: '<S2>/min_sat'
       *  Sum: '<S2>/Sum4'
       */
      rtb_Switch1 = 0.0 - reg_FF_PI_pl_regr_stiff_B->Input15;
    } else {
      rtb_Switch1 = rtb_Sum_d;
    }

    /* End of Switch: '<S103>/Switch2' */
  } else {
    rtb_Switch1 = 0.0;
  }

  /* End of Switch: '<Root>/Switch' */

  /* MATLAB Function: '<S1>/MATLAB Function' incorporates:
   *  Constant: '<S1>/Constant3'
   */
  tmp[0] = AlphaX;
  tmp[1] = AlphaY;
  tmp[2] = HTransform_tmp;
  tmp[3] = HTransform_tmp_0;
  tmp[4] = tmp_b;
  tmp[5] = tmp_c;
  tmp[6] = reg_FF_PI_pl_regr_stiff_B->Input15;
  tmp[7] = 1.0F;
  tmp_5 = 0.0F;
  for (i = 0; i < 8; i++) {
    tmp_5 += (real32_T)reg_FF_PI_pl_regr_stiff_ConstP.Constant3_Value[6 * i] *
      tmp[i];
  }

  tmp[0] = AlphaX;
  tmp[1] = AlphaY;
  tmp[2] = HTransform_tmp;
  tmp[3] = HTransform_tmp_0;
  tmp[4] = tmp_b;
  tmp[5] = tmp_c;
  tmp[6] = reg_FF_PI_pl_regr_stiff_B->Input15;
  tmp[7] = 1.0F;
  tmp_6 = 0.0F;
  for (i = 0; i < 8; i++) {
    tmp_6 += (real32_T)reg_FF_PI_pl_regr_stiff_ConstP.Constant3_Value[6 * i + 1]
      * tmp[i];
  }

  tmp[0] = AlphaX;
  tmp[1] = AlphaY;
  tmp[2] = HTransform_tmp;
  tmp[3] = HTransform_tmp_0;
  tmp[4] = tmp_b;
  tmp[5] = tmp_c;
  tmp[6] = reg_FF_PI_pl_regr_stiff_B->Input15;
  tmp[7] = 1.0F;
  tmp_7 = 0.0F;
  for (i = 0; i < 8; i++) {
    tmp_7 += (real32_T)reg_FF_PI_pl_regr_stiff_ConstP.Constant3_Value[6 * i + 2]
      * tmp[i];
  }

  tmp[0] = AlphaX;
  tmp[1] = AlphaY;
  tmp[2] = HTransform_tmp;
  tmp[3] = HTransform_tmp_0;
  tmp[4] = tmp_b;
  tmp[5] = tmp_c;
  tmp[6] = reg_FF_PI_pl_regr_stiff_B->Input15;
  tmp[7] = 1.0F;
  tmp_8 = 0.0F;
  for (i = 0; i < 8; i++) {
    tmp_8 += (real32_T)reg_FF_PI_pl_regr_stiff_ConstP.Constant3_Value[6 * i + 3]
      * tmp[i];
  }

  tmp[0] = AlphaX;
  tmp[1] = AlphaY;
  tmp[2] = HTransform_tmp;
  tmp[3] = HTransform_tmp_0;
  tmp[4] = tmp_b;
  tmp[5] = tmp_c;
  tmp[6] = reg_FF_PI_pl_regr_stiff_B->Input15;
  tmp[7] = 1.0F;
  tmp_9 = 0.0F;
  for (i = 0; i < 8; i++) {
    tmp_9 += (real32_T)reg_FF_PI_pl_regr_stiff_ConstP.Constant3_Value[6 * i + 4]
      * tmp[i];
  }

  tmp[0] = AlphaX;
  tmp[1] = AlphaY;
  tmp[2] = HTransform_tmp;
  tmp[3] = HTransform_tmp_0;
  tmp[4] = tmp_b;
  tmp[5] = tmp_c;
  tmp[6] = reg_FF_PI_pl_regr_stiff_B->Input15;
  tmp[7] = 1.0F;
  tmp_a = 0.0F;
  for (i = 0; i < 8; i++) {
    tmp_a += (real32_T)reg_FF_PI_pl_regr_stiff_ConstP.Constant3_Value[6 * i + 5]
      * tmp[i];
  }

  tmp_0[0] = tmp_5;
  tmp_0[1] = tmp_6;
  tmp_0[2] = tmp_7;
  tmp_0[3] = tmp_8;
  tmp_0[4] = tmp_9;
  tmp_0[5] = tmp_a;
  tmp_1[0] = 1.0F;
  tmp_1[1] = reg_FF_PI_pl_regr_stiff_B->Input1;
  tmp_1[2] = reg_FF_PI_pl_regr_stiff_B->Input2;
  tmp_1[3] = tmp_2;
  tmp_1[4] = tmp_3;
  tmp_1[5] = tmp_4;
  tmp_5 = 0.0F;
  for (i = 0; i < 6; i++) {
    tmp_5 += tmp_0[i] * tmp_1[i];
  }

  /* Sum: '<Root>/Sum2' incorporates:
   *  MATLAB Function: '<S1>/MATLAB Function'
   */
  reg_FF_PI_pl_regr_stiff_B->Sum2 = (real32_T)(rtb_Switch1 + tmp_5);

  /* S-Function (bur_out): '<Root>/Output2' */
  inst->Yellow_tab = reg_FF_PI_pl_regr_stiff_B->Sum2;

  /* MATLAB Function: '<S4>/requested alfa 2 deltaz1' */
  for (i = 0; i < 4; i++) {
    Green0_tmp_tmp_0[i] = (real32_T)Blue0_tmp[i] - ((HTransform[i + 4] *
      -73.6121597F + HTransform[i] * -42.5F) + HTransform[i + 12]);
  }

  /* Sum: '<S2>/Sum1' incorporates:
   *  Constant: '<S12>/cylinder height'
   *  Constant: '<S9>/cylinder height'
   *  Gain: '<S4>/Gain2'
   *  Gain: '<S4>/Gain5'
   *  MATLAB Function: '<S4>/requested alfa 2 deltaz1'
   *  Sum: '<S12>/Sum'
   *  Sum: '<S9>/Sum'
   */
  rtb_Sum1 = (0.001F * reg_FF_PI_pl_regr_stiff_norm(Green0_tmp_tmp_0, inst) - 0.115) -
    (0.001F * reg_FF_PI_pl_regr_stiff_norm(Blue0_tmp_0, inst) - 0.115);

  /* S-Function (bur_in): '<Root>/Input6' */
  reg_FF_PI_pl_regr_stiff_B->Input6 = inst->reset_PID_yellow;

  /* DiscreteIntegrator: '<S46>/Integrator' */
  if ((reg_FF_PI_pl_regr_stiff_B->Input6 <= 0.0F) &&
      (reg_FF_PI_pl_regr_stiff_DW->Integrator_PrevResetState_e == 1)) {
    reg_FF_PI_pl_regr_stiff_DW->Integrator_DSTATE_i = 0.0;
  }

  /* DiscreteIntegrator: '<S41>/Filter' */
  if ((reg_FF_PI_pl_regr_stiff_B->Input6 <= 0.0F) &&
      (reg_FF_PI_pl_regr_stiff_DW->Filter_PrevResetState_h == 1)) {
    reg_FF_PI_pl_regr_stiff_DW->Filter_DSTATE_a = 0.0;
  }

  /* Product: '<S49>/NProd Out' incorporates:
   *  DiscreteIntegrator: '<S41>/Filter'
   *  Product: '<S40>/DProd Out'
   *  Sum: '<S41>/SumD'
   */
  rtb_Sum_d = (rtb_Sum1 * reg_FF_PI_pl_regr_stiff_B->Input13 -
               reg_FF_PI_pl_regr_stiff_DW->Filter_DSTATE_a) *
    reg_FF_PI_pl_regr_stiff_B->Input14;

  /* Switch: '<Root>/Switch1' */
  if (reg_FF_PI_pl_regr_stiff_B->Input6 > 0.0F) {
    /* Sum: '<S56>/Sum' incorporates:
     *  DiscreteIntegrator: '<S46>/Integrator'
     *  Product: '<S51>/PProd Out'
     */
    rtb_Switch1 = (rtb_Sum1 * reg_FF_PI_pl_regr_stiff_B->Input11 +
                   reg_FF_PI_pl_regr_stiff_DW->Integrator_DSTATE_i) + rtb_Sum_d;

    /* Switch: '<S54>/Switch2' incorporates:
     *  Constant: '<S2>/max_sat'
     *  Constant: '<S2>/min_sat'
     *  RelationalOperator: '<S54>/LowerRelop1'
     *  RelationalOperator: '<S54>/UpperRelop'
     *  Sum: '<S2>/Sum3'
     *  Sum: '<S2>/Sum4'
     *  Switch: '<S54>/Switch'
     */
    if (rtb_Switch1 > 5.0 - reg_FF_PI_pl_regr_stiff_B->Input15) {
      rtb_Switch1 = 5.0 - reg_FF_PI_pl_regr_stiff_B->Input15;
    } else if (rtb_Switch1 < 0.0 - reg_FF_PI_pl_regr_stiff_B->Input15) {
      /* Switch: '<S54>/Switch' incorporates:
       *  Constant: '<S2>/min_sat'
       *  Sum: '<S2>/Sum4'
       */
      rtb_Switch1 = 0.0 - reg_FF_PI_pl_regr_stiff_B->Input15;
    }

    /* End of Switch: '<S54>/Switch2' */
  } else {
    rtb_Switch1 = 0.0;
  }

  /* End of Switch: '<Root>/Switch1' */

  /* MATLAB Function: '<S1>/MATLAB Function' incorporates:
   *  Constant: '<S1>/Constant1'
   */
  tmp[0] = AlphaX;
  tmp[1] = AlphaY;
  tmp[2] = HTransform_tmp;
  tmp[3] = HTransform_tmp_0;
  tmp[4] = tmp_b;
  tmp[5] = tmp_c;
  tmp[6] = reg_FF_PI_pl_regr_stiff_B->Input15;
  tmp[7] = 1.0F;
  tmp_5 = 0.0F;
  for (i = 0; i < 8; i++) {
    tmp_5 += (real32_T)reg_FF_PI_pl_regr_stiff_ConstP.Constant1_Value[6 * i] *
      tmp[i];
  }

  tmp[0] = AlphaX;
  tmp[1] = AlphaY;
  tmp[2] = HTransform_tmp;
  tmp[3] = HTransform_tmp_0;
  tmp[4] = tmp_b;
  tmp[5] = tmp_c;
  tmp[6] = reg_FF_PI_pl_regr_stiff_B->Input15;
  tmp[7] = 1.0F;
  tmp_6 = 0.0F;
  for (i = 0; i < 8; i++) {
    tmp_6 += (real32_T)reg_FF_PI_pl_regr_stiff_ConstP.Constant1_Value[6 * i + 1]
      * tmp[i];
  }

  tmp[0] = AlphaX;
  tmp[1] = AlphaY;
  tmp[2] = HTransform_tmp;
  tmp[3] = HTransform_tmp_0;
  tmp[4] = tmp_b;
  tmp[5] = tmp_c;
  tmp[6] = reg_FF_PI_pl_regr_stiff_B->Input15;
  tmp[7] = 1.0F;
  tmp_7 = 0.0F;
  for (i = 0; i < 8; i++) {
    tmp_7 += (real32_T)reg_FF_PI_pl_regr_stiff_ConstP.Constant1_Value[6 * i + 2]
      * tmp[i];
  }

  tmp[0] = AlphaX;
  tmp[1] = AlphaY;
  tmp[2] = HTransform_tmp;
  tmp[3] = HTransform_tmp_0;
  tmp[4] = tmp_b;
  tmp[5] = tmp_c;
  tmp[6] = reg_FF_PI_pl_regr_stiff_B->Input15;
  tmp[7] = 1.0F;
  tmp_8 = 0.0F;
  for (i = 0; i < 8; i++) {
    tmp_8 += (real32_T)reg_FF_PI_pl_regr_stiff_ConstP.Constant1_Value[6 * i + 3]
      * tmp[i];
  }

  tmp[0] = AlphaX;
  tmp[1] = AlphaY;
  tmp[2] = HTransform_tmp;
  tmp[3] = HTransform_tmp_0;
  tmp[4] = tmp_b;
  tmp[5] = tmp_c;
  tmp[6] = reg_FF_PI_pl_regr_stiff_B->Input15;
  tmp[7] = 1.0F;
  tmp_9 = 0.0F;
  for (i = 0; i < 8; i++) {
    tmp_9 += (real32_T)reg_FF_PI_pl_regr_stiff_ConstP.Constant1_Value[6 * i + 4]
      * tmp[i];
  }

  tmp[0] = AlphaX;
  tmp[1] = AlphaY;
  tmp[2] = HTransform_tmp;
  tmp[3] = HTransform_tmp_0;
  tmp[4] = tmp_b;
  tmp[5] = tmp_c;
  tmp[6] = reg_FF_PI_pl_regr_stiff_B->Input15;
  tmp[7] = 1.0F;
  AlphaX = 0.0F;
  for (i = 0; i < 8; i++) {
    AlphaX += (real32_T)reg_FF_PI_pl_regr_stiff_ConstP.Constant1_Value[6 * i + 5]
      * tmp[i];
  }

  tmp_0[0] = tmp_5;
  tmp_0[1] = tmp_6;
  tmp_0[2] = tmp_7;
  tmp_0[3] = tmp_8;
  tmp_0[4] = tmp_9;
  tmp_0[5] = AlphaX;
  tmp_1[0] = 1.0F;
  tmp_1[1] = reg_FF_PI_pl_regr_stiff_B->Input1;
  tmp_1[2] = reg_FF_PI_pl_regr_stiff_B->Input2;
  tmp_1[3] = tmp_2;
  tmp_1[4] = tmp_3;
  tmp_1[5] = tmp_4;
  AlphaX = 0.0F;
  for (i = 0; i < 6; i++) {
    AlphaX += tmp_0[i] * tmp_1[i];
  }

  /* Sum: '<Root>/Sum1' incorporates:
   *  MATLAB Function: '<S1>/MATLAB Function'
   */
  reg_FF_PI_pl_regr_stiff_B->Sum1 = (real32_T)(rtb_Switch1 + AlphaX);

  /* S-Function (bur_out): '<Root>/Output4' */
  inst->Green_tab = reg_FF_PI_pl_regr_stiff_B->Sum1;

  /* S-Function (bur_in): '<Root>/Input10' */
  reg_FF_PI_pl_regr_stiff_B->Input10 = inst->tlak3;

  /* S-Function (bur_in): '<Root>/Input12' */
  reg_FF_PI_pl_regr_stiff_B->Input12 = inst->I_parameter;

  /* S-Function (bur_in): '<Root>/Input8' */
  reg_FF_PI_pl_regr_stiff_B->Input8 = inst->tlak1;

  /* S-Function (bur_in): '<Root>/Input9' */
  reg_FF_PI_pl_regr_stiff_B->Input9 = inst->tlak2;

  /* Product: '<S43>/IProd Out' */
  rtb_Switch1 = rtb_Sum1 * reg_FF_PI_pl_regr_stiff_B->Input12;

  /* Product: '<S92>/IProd Out' */
  rtb_Sum2 *= reg_FF_PI_pl_regr_stiff_B->Input12;

  /* Product: '<S141>/IProd Out' */
  A2 *= reg_FF_PI_pl_regr_stiff_B->Input12;

  /* Update for DiscreteIntegrator: '<S144>/Integrator' */
  reg_FF_PI_pl_regr_stiff_DW->Integrator_DSTATE += 0.002 * A2;
  if (reg_FF_PI_pl_regr_stiff_B->Input5 > 0.0F) {
    reg_FF_PI_pl_regr_stiff_DW->Integrator_PrevResetState = 1;
  } else if (reg_FF_PI_pl_regr_stiff_B->Input5 < 0.0F) {
    reg_FF_PI_pl_regr_stiff_DW->Integrator_PrevResetState = -1;
  } else if (reg_FF_PI_pl_regr_stiff_B->Input5 == 0.0F) {
    reg_FF_PI_pl_regr_stiff_DW->Integrator_PrevResetState = 0;
  } else {
    reg_FF_PI_pl_regr_stiff_DW->Integrator_PrevResetState = 2;
  }

  /* End of Update for DiscreteIntegrator: '<S144>/Integrator' */

  /* Update for DiscreteIntegrator: '<S139>/Filter' */
  reg_FF_PI_pl_regr_stiff_DW->Filter_DSTATE += 0.002 * A1;
  if (reg_FF_PI_pl_regr_stiff_B->Input5 > 0.0F) {
    reg_FF_PI_pl_regr_stiff_DW->Filter_PrevResetState = 1;
  } else if (reg_FF_PI_pl_regr_stiff_B->Input5 < 0.0F) {
    reg_FF_PI_pl_regr_stiff_DW->Filter_PrevResetState = -1;
  } else if (reg_FF_PI_pl_regr_stiff_B->Input5 == 0.0F) {
    reg_FF_PI_pl_regr_stiff_DW->Filter_PrevResetState = 0;
  } else {
    reg_FF_PI_pl_regr_stiff_DW->Filter_PrevResetState = 2;
  }

  /* End of Update for DiscreteIntegrator: '<S139>/Filter' */

  /* Update for DiscreteIntegrator: '<S95>/Integrator' */
  reg_FF_PI_pl_regr_stiff_DW->Integrator_DSTATE_o += 0.002 * rtb_Sum2;
  if (reg_FF_PI_pl_regr_stiff_B->Input7 > 0.0F) {
    reg_FF_PI_pl_regr_stiff_DW->Integrator_PrevResetState_l = 1;
  } else if (reg_FF_PI_pl_regr_stiff_B->Input7 < 0.0F) {
    reg_FF_PI_pl_regr_stiff_DW->Integrator_PrevResetState_l = -1;
  } else if (reg_FF_PI_pl_regr_stiff_B->Input7 == 0.0F) {
    reg_FF_PI_pl_regr_stiff_DW->Integrator_PrevResetState_l = 0;
  } else {
    reg_FF_PI_pl_regr_stiff_DW->Integrator_PrevResetState_l = 2;
  }

  /* End of Update for DiscreteIntegrator: '<S95>/Integrator' */

  /* Update for DiscreteIntegrator: '<S90>/Filter' */
  reg_FF_PI_pl_regr_stiff_DW->Filter_DSTATE_f += 0.002 * A3;
  if (reg_FF_PI_pl_regr_stiff_B->Input7 > 0.0F) {
    reg_FF_PI_pl_regr_stiff_DW->Filter_PrevResetState_e = 1;
  } else if (reg_FF_PI_pl_regr_stiff_B->Input7 < 0.0F) {
    reg_FF_PI_pl_regr_stiff_DW->Filter_PrevResetState_e = -1;
  } else if (reg_FF_PI_pl_regr_stiff_B->Input7 == 0.0F) {
    reg_FF_PI_pl_regr_stiff_DW->Filter_PrevResetState_e = 0;
  } else {
    reg_FF_PI_pl_regr_stiff_DW->Filter_PrevResetState_e = 2;
  }

  /* End of Update for DiscreteIntegrator: '<S90>/Filter' */

  /* Update for DiscreteIntegrator: '<S46>/Integrator' */
  reg_FF_PI_pl_regr_stiff_DW->Integrator_DSTATE_i += 0.002 * rtb_Switch1;
  if (reg_FF_PI_pl_regr_stiff_B->Input6 > 0.0F) {
    reg_FF_PI_pl_regr_stiff_DW->Integrator_PrevResetState_e = 1;
  } else if (reg_FF_PI_pl_regr_stiff_B->Input6 < 0.0F) {
    reg_FF_PI_pl_regr_stiff_DW->Integrator_PrevResetState_e = -1;
  } else if (reg_FF_PI_pl_regr_stiff_B->Input6 == 0.0F) {
    reg_FF_PI_pl_regr_stiff_DW->Integrator_PrevResetState_e = 0;
  } else {
    reg_FF_PI_pl_regr_stiff_DW->Integrator_PrevResetState_e = 2;
  }

  /* End of Update for DiscreteIntegrator: '<S46>/Integrator' */

  /* Update for DiscreteIntegrator: '<S41>/Filter' */
  reg_FF_PI_pl_regr_stiff_DW->Filter_DSTATE_a += 0.002 * rtb_Sum_d;
  if (reg_FF_PI_pl_regr_stiff_B->Input6 > 0.0F) {
    reg_FF_PI_pl_regr_stiff_DW->Filter_PrevResetState_h = 1;
  } else if (reg_FF_PI_pl_regr_stiff_B->Input6 < 0.0F) {
    reg_FF_PI_pl_regr_stiff_DW->Filter_PrevResetState_h = -1;
  } else if (reg_FF_PI_pl_regr_stiff_B->Input6 == 0.0F) {
    reg_FF_PI_pl_regr_stiff_DW->Filter_PrevResetState_h = 0;
  } else {
    reg_FF_PI_pl_regr_stiff_DW->Filter_PrevResetState_h = 2;
  }

  /* End of Update for DiscreteIntegrator: '<S41>/Filter' */
}

/* Model initialize function */
void reg_FF_PI_pl_regr_stiff_initialize(RT_MODEL_reg_FF_PI_pl_regr_st_T *const
  reg_FF_PI_pl_regr_stiff_M, struct FF_PID_r_t* inst)
{
  DW_reg_FF_PI_pl_regr_stiff_T *reg_FF_PI_pl_regr_stiff_DW =
    reg_FF_PI_pl_regr_stiff_M->dwork;

  /* InitializeConditions for DiscreteIntegrator: '<S144>/Integrator' */
  reg_FF_PI_pl_regr_stiff_DW->Integrator_DSTATE = 0.0;
  reg_FF_PI_pl_regr_stiff_DW->Integrator_PrevResetState = 2;

  /* InitializeConditions for DiscreteIntegrator: '<S139>/Filter' */
  reg_FF_PI_pl_regr_stiff_DW->Filter_DSTATE = 0.0;
  reg_FF_PI_pl_regr_stiff_DW->Filter_PrevResetState = 2;

  /* InitializeConditions for DiscreteIntegrator: '<S95>/Integrator' */
  reg_FF_PI_pl_regr_stiff_DW->Integrator_DSTATE_o = 0.0;
  reg_FF_PI_pl_regr_stiff_DW->Integrator_PrevResetState_l = 2;

  /* InitializeConditions for DiscreteIntegrator: '<S90>/Filter' */
  reg_FF_PI_pl_regr_stiff_DW->Filter_DSTATE_f = 0.0;
  reg_FF_PI_pl_regr_stiff_DW->Filter_PrevResetState_e = 2;

  /* InitializeConditions for DiscreteIntegrator: '<S46>/Integrator' */
  reg_FF_PI_pl_regr_stiff_DW->Integrator_DSTATE_i = 0.0;
  reg_FF_PI_pl_regr_stiff_DW->Integrator_PrevResetState_e = 2;

  /* InitializeConditions for DiscreteIntegrator: '<S41>/Filter' */
  reg_FF_PI_pl_regr_stiff_DW->Filter_DSTATE_a = 0.0;
  reg_FF_PI_pl_regr_stiff_DW->Filter_PrevResetState_h = 2;
}

/* Model terminate function */
void reg_FF_PI_pl_regr_stiff_terminate(RT_MODEL_reg_FF_PI_pl_regr_st_T
  * reg_FF_PI_pl_regr_stiff_M, struct FF_PID_r_t* inst)
{}

/* Model data allocation function */
void reg_FF_PI_pl_regr_stiff_initializeMemory(RT_MODEL_reg_FF_PI_pl_regr_st_T* const reg_FF_PI_pl_regr_stiff_M, struct FF_PID_r_t * inst)
{  /* states (dwork) */
  {
  }

  {
    B_reg_FF_PI_pl_regr_stiff_T *reg_FF_PI_pl_regr_stiff_B =
      reg_FF_PI_pl_regr_stiff_M->blockIO;
    DW_reg_FF_PI_pl_regr_stiff_T *reg_FF_PI_pl_regr_stiff_DW =
      reg_FF_PI_pl_regr_stiff_M->dwork;

    /* block I/O */
    {
      reg_FF_PI_pl_regr_stiff_B->Input15 = 0.0F;
      reg_FF_PI_pl_regr_stiff_B->Input1 = 0.0F;
      reg_FF_PI_pl_regr_stiff_B->Input2 = 0.0F;
      reg_FF_PI_pl_regr_stiff_B->Input3 = 0.0F;
      reg_FF_PI_pl_regr_stiff_B->Input4 = 0.0F;
      reg_FF_PI_pl_regr_stiff_B->Input11 = 0.0F;
      reg_FF_PI_pl_regr_stiff_B->Input5 = 0.0F;
      reg_FF_PI_pl_regr_stiff_B->Input13 = 0.0F;
      reg_FF_PI_pl_regr_stiff_B->Input14 = 0.0F;
      reg_FF_PI_pl_regr_stiff_B->Sum = 0.0F;
      reg_FF_PI_pl_regr_stiff_B->Input7 = 0.0F;
      reg_FF_PI_pl_regr_stiff_B->Sum2 = 0.0F;
      reg_FF_PI_pl_regr_stiff_B->Input6 = 0.0F;
      reg_FF_PI_pl_regr_stiff_B->Sum1 = 0.0F;
      reg_FF_PI_pl_regr_stiff_B->Input10 = 0.0F;
      reg_FF_PI_pl_regr_stiff_B->Input12 = 0.0F;
      reg_FF_PI_pl_regr_stiff_B->Input8 = 0.0F;
      reg_FF_PI_pl_regr_stiff_B->Input9 = 0.0F;
    }

    /* states (dwork) */
    (void) memset((void *)reg_FF_PI_pl_regr_stiff_DW, 0,
                  sizeof(DW_reg_FF_PI_pl_regr_stiff_T));
    reg_FF_PI_pl_regr_stiff_DW->Integrator_DSTATE = 0.0;
    reg_FF_PI_pl_regr_stiff_DW->Filter_DSTATE = 0.0;
    reg_FF_PI_pl_regr_stiff_DW->Integrator_DSTATE_o = 0.0;
    reg_FF_PI_pl_regr_stiff_DW->Filter_DSTATE_f = 0.0;
    reg_FF_PI_pl_regr_stiff_DW->Integrator_DSTATE_i = 0.0;
    reg_FF_PI_pl_regr_stiff_DW->Filter_DSTATE_a = 0.0;
  }

}
```

### Library Logical/Libraries/traj_lib (ANSIC, version 1.00.0)

#### generator_trajektorie_test.c
```c
/*
 * generator_trajektorie_test.c
 *
 * Academic License - for use in teaching, academic research, and meeting
 * course requirements at degree granting institutions only.  Not for
 * government, commercial, or other organizational use.
 *
 * Code generation for model "generator_trajektorie_test".
 *
 * Model version              : 1.23
 * Simulink Coder version : 9.6 (R2021b) 14-May-2021
 * C source code generated on : Fri Mar 25 13:28:48 2022
 *
 * Target selection: bur_grt.tlc
 * Note: GRT includes extra infrastructure and instrumentation for prototyping
 * Embedded hardware selection: Intel->x86/Pentium
 * Code generation objectives: Unspecified
 * Validation result: Not run
 */

#include "generator_trajektorie_test.h"
#include "generator_trajektorie_test_private.h"

/* Model step function */
void generator_trajektorie_test_step(RT_MODEL_generator_trajektori_T *const
  generator_trajektorie_test_M, struct traj* inst)
{
  B_generator_trajektorie_test_T *generator_trajektorie_test_B =
    generator_trajektorie_test_M->blockIO;
  real_T rtb_usecka[300];
  real_T par_funkcie[100];
  real_T pocitadlo;
  int32_T b_poradie_0_1;
  int32_T i;
  real32_T a_tmp;
  real32_T b;
  real32_T b_a_tmp;
  real32_T cas_pohybu;
  real32_T pocet_skokov;
  real32_T tmp;
  boolean_T exitg1;

  /* S-Function (bur_in): '<Root>/Input1' */
  generator_trajektorie_test_B->Input1 = inst->aktualny_uhol_x;

  /* S-Function (bur_in): '<Root>/Input2' */
  generator_trajektorie_test_B->Input2 = inst->aktualny_uhol_y;

  /* S-Function (bur_in): '<Root>/Input3' */
  generator_trajektorie_test_B->Input3 = inst->pozadovany_uhol_x;

  /* S-Function (bur_in): '<Root>/Input4' */
  generator_trajektorie_test_B->Input4 = inst->pozadovany_uhol_y;

  /* S-Function (bur_in): '<Root>/Input' */
  generator_trajektorie_test_B->Input = inst->dlzka_pohybu;

  /* MATLAB Function: '<Root>/MATLAB Function' incorporates:
   *  SignalConversion generated from: '<S1>/ SFunction '
   */
  a_tmp = generator_trajektorie_test_B->Input3 -
    generator_trajektorie_test_B->Input1;
  b_a_tmp = generator_trajektorie_test_B->Input4 -
    generator_trajektorie_test_B->Input2;
  pocet_skokov = sqrtf(a_tmp * a_tmp + b_a_tmp * b_a_tmp);
  cas_pohybu = pocet_skokov * generator_trajektorie_test_B->Input / 42.4264107F;
  pocitadlo = 0.0;
  pocet_skokov = ceilf(pocet_skokov * 99.0F / 56.5685387F);
  for (i = 0; i < 100; i++) {
    par_funkcie[i] = 0.0;
  }

  for (i = 0; i < 300; i++) {
    rtb_usecka[i] = 0.0;
  }

  b = 1.0F / pocet_skokov;
  i = (int32_T)(((b - -0.5F) + 0.5F) / b);
  for (b_poradie_0_1 = 0; b_poradie_0_1 < i; b_poradie_0_1++) {
    real32_T poradie_0_1;
    poradie_0_1 = (real32_T)b_poradie_0_1 * b + -0.5F;
    pocitadlo++;
    tmp = fabsf(poradie_0_1);
    if (poradie_0_1 < 0.0F) {
      poradie_0_1 = -1.0F;
    } else if (poradie_0_1 > 0.0F) {
      poradie_0_1 = 1.0F;
    } else if (poradie_0_1 == 0.0F) {
      poradie_0_1 = 0.0F;
    } else {
      poradie_0_1 = (rtNaNF);
    }

    par_funkcie[(int32_T)pocitadlo - 1] = (poradie_0_1 * 4.0F * tmp * (1.0F -
      tmp) + 1.0F) / 2.0F;
  }

  i = 0;
  exitg1 = false;
  while ((!exitg1) && (i < 100)) {
    rtb_usecka[3 * i] = a_tmp * (real32_T)par_funkcie[i] +
      generator_trajektorie_test_B->Input1;
    rtb_usecka[3 * i + 1] = b_a_tmp * (real32_T)par_funkcie[i] +
      generator_trajektorie_test_B->Input2;
    rtb_usecka[3 * i + 2] = (((real32_T)i + 1.0F) - 1.0F) * cas_pohybu /
      (pocet_skokov + 1.0F);
    if ((real_T)i + 1.0 == pocet_skokov + 1.0F) {
      exitg1 = true;
    } else {
      i++;
    }
  }

  for (i = 0; i < 300; i++) {
    /* Gain: '<Root>/Gain' */
    generator_trajektorie_test_B->Gain[i] = (real32_T)rtb_usecka[i];
  }

  /* S-Function (bur_out): '<Root>/Output' */
  {
    real32_T *u1 = &inst->trajektoria
      [0]
      [0];

    {
      int_T i1;
      const real32_T *u0 = &generator_trajektorie_test_B->Gain[0];
      for (i1=0; i1 < 300; i1++) {
        u1[i1] = u0[i1];
      }
    }
  }

  /* MATLAB Function: '<Root>/MATLAB Function' */
  if (rtIsNaNF(pocet_skokov + 1.0F) || rtIsInfF(pocet_skokov + 1.0F)) {
    tmp = 0.0F;
  } else {
    tmp = fmodf(pocet_skokov + 1.0F, 65536.0F);
  }

  /* Gain: '<Root>/Gain1' incorporates:
   *  MATLAB Function: '<Root>/MATLAB Function'
   */
  generator_trajektorie_test_B->Gain1 = (int16_T)(tmp < 0.0F ? (int32_T)(int16_T)
    -(int16_T)(uint16_T)-tmp : (int32_T)(int16_T)(uint16_T)tmp);

  /* S-Function (bur_out): '<Root>/Output1' */
  inst->pocet_bodov_traj = generator_trajektorie_test_B->Gain1;
}

/* Model initialize function */
void generator_trajektorie_test_initialize(RT_MODEL_generator_trajektori_T *
  const generator_trajektorie_test_M, struct traj* inst)
{
  UNUSED_PARAMETER(generator_trajektorie_test_M);
}

/* Model terminate function */
void generator_trajektorie_test_terminate(RT_MODEL_generator_trajektori_T
  * generator_trajektorie_test_M, struct traj* inst)
{}

/* Model data allocation function */
void generator_trajektorie_test_initializeMemory(RT_MODEL_generator_trajektori_T* const generator_trajektorie_test_M, struct traj * inst)
{
  /* block I/O */
  {
  }

  {
    B_generator_trajektorie_test_T *generator_trajektorie_test_B =
      generator_trajektorie_test_M->blockIO;

    /* initialize non-finites */
    rt_InitInfAndNaN(sizeof(real_T));

    /* block I/O */
    (void) memset(((void *) generator_trajektorie_test_B), 0,
                  sizeof(B_generator_trajektorie_test_T));

    {
      int32_T i;
      for (i = 0; i < 300; i++) {
        generator_trajektorie_test_B->Gain[i] = 0.0F;
      }

      generator_trajektorie_test_B->Input1 = 0.0F;
      generator_trajektorie_test_B->Input2 = 0.0F;
      generator_trajektorie_test_B->Input3 = 0.0F;
      generator_trajektorie_test_B->Input4 = 0.0F;
      generator_trajektorie_test_B->Input = 0.0F;
    }
  }

}
```

#### rtGetInf.c
```c
/*
 * rtGetInf.c
 *
 * Academic License - for use in teaching, academic research, and meeting
 * course requirements at degree granting institutions only.  Not for
 * government, commercial, or other organizational use.
 *
 * Code generation for model "generator_trajektorie_test".
 *
 * Model version              : 1.23
 * Simulink Coder version : 9.6 (R2021b) 14-May-2021
 * C source code generated on : Fri Mar 25 13:28:48 2022
 *
 * Target selection: bur_grt.tlc
 * Note: GRT includes extra infrastructure and instrumentation for prototyping
 * Embedded hardware selection: Intel->x86/Pentium
 * Code generation objectives: Unspecified
 * Validation result: Not run
 */

/*
 * Abstract:
 *      Function to initialize non-finite, Inf
 */
#include "rtGetInf.h"
#define NumBitsPerChar                 8U

/*
 * Initialize rtInf needed by the generated code.
 * Inf is initialized as non-signaling. Assumes IEEE.
 */
real_T rtGetInf(void)
{
  size_t bitsPerReal = sizeof(real_T) * (NumBitsPerChar);
  real_T inf = 0.0;
  if (bitsPerReal == 32U) {
    inf = rtGetInfF();
  } else {
    uint16_T one = 1U;
    enum {
      LittleEndian,
      BigEndian
    } machByteOrder = (*((uint8_T *) &one) == 1U) ? LittleEndian : BigEndian;
    switch (machByteOrder) {
     case LittleEndian:
      {
        union {
          LittleEndianIEEEDouble bitVal;
          real_T fltVal;
        } tmpVal;

        tmpVal.bitVal.words.wordH = 0x7FF00000U;
        tmpVal.bitVal.words.wordL = 0x00000000U;
        inf = tmpVal.fltVal;
        break;
      }

     case BigEndian:
      {
        union {
          BigEndianIEEEDouble bitVal;
          real_T fltVal;
        } tmpVal;

        tmpVal.bitVal.words.wordH = 0x7FF00000U;
        tmpVal.bitVal.words.wordL = 0x00000000U;
        inf = tmpVal.fltVal;
        break;
      }
    }
  }

  return inf;
}

/*
 * Initialize rtInfF needed by the generated code.
 * Inf is initialized as non-signaling. Assumes IEEE.
 */
real32_T rtGetInfF(void)
{
  IEEESingle infF;
  infF.wordL.wordLuint = 0x7F800000U;
  return infF.wordL.wordLreal;
}

/*
 * Initialize rtMinusInf needed by the generated code.
 * Inf is initialized as non-signaling. Assumes IEEE.
 */
real_T rtGetMinusInf(void)
{
  size_t bitsPerReal = sizeof(real_T) * (NumBitsPerChar);
  real_T minf = 0.0;
  if (bitsPerReal == 32U) {
    minf = rtGetMinusInfF();
  } else {
    uint16_T one = 1U;
    enum {
      LittleEndian,
      BigEndian
    } machByteOrder = (*((uint8_T *) &one) == 1U) ? LittleEndian : BigEndian;
    switch (machByteOrder) {
     case LittleEndian:
      {
        union {
          LittleEndianIEEEDouble bitVal;
          real_T fltVal;
        } tmpVal;

        tmpVal.bitVal.words.wordH = 0xFFF00000U;
        tmpVal.bitVal.words.wordL = 0x00000000U;
        minf = tmpVal.fltVal;
        break;
      }

     case BigEndian:
      {
        union {
          BigEndianIEEEDouble bitVal;
          real_T fltVal;
        } tmpVal;

        tmpVal.bitVal.words.wordH = 0xFFF00000U;
        tmpVal.bitVal.words.wordL = 0x00000000U;
        minf = tmpVal.fltVal;
        break;
      }
    }
  }

  return minf;
}

/*
 * Initialize rtMinusInfF needed by the generated code.
 * Inf is initialized as non-signaling. Assumes IEEE.
 */
real32_T rtGetMinusInfF(void)
{
  IEEESingle minfF;
  minfF.wordL.wordLuint = 0xFF800000U;
  return minfF.wordL.wordLreal;
}
```

#### rtGetNaN.h
```c
/*
 * rtGetNaN.h
 *
 * Academic License - for use in teaching, academic research, and meeting
 * course requirements at degree granting institutions only.  Not for
 * government, commercial, or other organizational use.
 *
 * Code generation for model "generator_trajektorie_test".
 *
 * Model version              : 1.23
 * Simulink Coder version : 9.6 (R2021b) 14-May-2021
 * C source code generated on : Fri Mar 25 13:28:48 2022
 *
 * Target selection: bur_grt.tlc
 * Note: GRT includes extra infrastructure and instrumentation for prototyping
 * Embedded hardware selection: Intel->x86/Pentium
 * Code generation objectives: Unspecified
 * Validation result: Not run
 */

#ifndef RTW_HEADER_rtGetNaN_h_
#define RTW_HEADER_rtGetNaN_h_
#include <stddef.h>
#include "rtwtypes.h"
#include "rt_nonfinite.h"

extern real_T rtGetNaN(void);
extern real32_T rtGetNaNF(void);

#endif                                 /* RTW_HEADER_rtGetNaN_h_ */
```

#### rt_nonfinite.c
```c
/*
 * rt_nonfinite.c
 *
 * Academic License - for use in teaching, academic research, and meeting
 * course requirements at degree granting institutions only.  Not for
 * government, commercial, or other organizational use.
 *
 * Code generation for model "generator_trajektorie_test".
 *
 * Model version              : 1.23
 * Simulink Coder version : 9.6 (R2021b) 14-May-2021
 * C source code generated on : Fri Mar 25 13:28:48 2022
 *
 * Target selection: bur_grt.tlc
 * Note: GRT includes extra infrastructure and instrumentation for prototyping
 * Embedded hardware selection: Intel->x86/Pentium
 * Code generation objectives: Unspecified
 * Validation result: Not run
 */

/*
 * Abstract:
 *      Function to initialize non-finites,
 *      (Inf, NaN and -Inf).
 */
#include "rt_nonfinite.h"
#include "rtGetNaN.h"
#include "rtGetInf.h"
#define NumBitsPerChar                 8U

real_T rtInf;
real_T rtMinusInf;
real_T rtNaN;
real32_T rtInfF;
real32_T rtMinusInfF;
real32_T rtNaNF;

/*
 * Initialize the rtInf, rtMinusInf, and rtNaN needed by the
 * generated code. NaN is initialized as non-signaling. Assumes IEEE.
 */
void rt_InitInfAndNaN(size_t realSize)
{
  (void) (realSize);
  rtNaN = rtGetNaN();
  rtNaNF = rtGetNaNF();
  rtInf = rtGetInf();
  rtInfF = rtGetInfF();
  rtMinusInf = rtGetMinusInf();
  rtMinusInfF = rtGetMinusInfF();
}

/* Test if value is infinite */
boolean_T rtIsInf(real_T value)
{
  return (boolean_T)((value==rtInf || value==rtMinusInf) ? 1U : 0U);
}

/* Test if single-precision value is infinite */
boolean_T rtIsInfF(real32_T value)
{
  return (boolean_T)(((value)==rtInfF || (value)==rtMinusInfF) ? 1U : 0U);
}

/* Test if value is not a number */
boolean_T rtIsNaN(real_T value)
{
  boolean_T result = (boolean_T) 0;
  size_t bitsPerReal = sizeof(real_T) * (NumBitsPerChar);
  if (bitsPerReal == 32U) {
    result = rtIsNaNF((real32_T)value);
  } else {
    union {
      LittleEndianIEEEDouble bitVal;
      real_T fltVal;
    } tmpVal;

    tmpVal.fltVal = value;
    result = (boolean_T)((tmpVal.bitVal.words.wordH & 0x7FF00000) == 0x7FF00000 &&
                         ( (tmpVal.bitVal.words.wordH & 0x000FFFFF) != 0 ||
                          (tmpVal.bitVal.words.wordL != 0) ));
  }

  return result;
}

/* Test if single-precision value is not a number */
boolean_T rtIsNaNF(real32_T value)
{
  IEEESingle tmp;
  tmp.wordL.wordLreal = value;
  return (boolean_T)( (tmp.wordL.wordLuint & 0x7F800000) == 0x7F800000 &&
                     (tmp.wordL.wordLuint & 0x007FFFFF) != 0 );
}
```

#### rt_nonfinite.h
```c
/*
 * rt_nonfinite.h
 *
 * Academic License - for use in teaching, academic research, and meeting
 * course requirements at degree granting institutions only.  Not for
 * government, commercial, or other organizational use.
 *
 * Code generation for model "generator_trajektorie_test".
 *
 * Model version              : 1.23
 * Simulink Coder version : 9.6 (R2021b) 14-May-2021
 * C source code generated on : Fri Mar 25 13:28:48 2022
 *
 * Target selection: bur_grt.tlc
 * Note: GRT includes extra infrastructure and instrumentation for prototyping
 * Embedded hardware selection: Intel->x86/Pentium
 * Code generation objectives: Unspecified
 * Validation result: Not run
 */

#ifndef RTW_HEADER_rt_nonfinite_h_
#define RTW_HEADER_rt_nonfinite_h_
#include <stddef.h>
#include "rtwtypes.h"

extern real_T rtInf;
extern real_T rtMinusInf;
extern real_T rtNaN;
extern real32_T rtInfF;
extern real32_T rtMinusInfF;
extern real32_T rtNaNF;
extern void rt_InitInfAndNaN(size_t realSize);
extern boolean_T rtIsInf(real_T value);
extern boolean_T rtIsInfF(real32_T value);
extern boolean_T rtIsNaN(real_T value);
extern boolean_T rtIsNaNF(real32_T value);
typedef struct {
  struct {
    uint32_T wordH;
    uint32_T wordL;
  } words;
} BigEndianIEEEDouble;

typedef struct {
  struct {
    uint32_T wordL;
    uint32_T wordH;
  } words;
} LittleEndianIEEEDouble;

typedef struct {
  union {
    real32_T wordLreal;
    uint32_T wordLuint;
  } wordL;
} IEEESingle;

#endif                                 /* RTW_HEADER_rt_nonfinite_h_ */
```

#### rtwtypes.h
```c
/*
 * rtwtypes.h
 *
 * Academic License - for use in teaching, academic research, and meeting
 * course requirements at degree granting institutions only.  Not for
 * government, commercial, or other organizational use.
 *
 * Code generation for model "generator_trajektorie_test".
 *
 * Model version              : 1.23
 * Simulink Coder version : 9.6 (R2021b) 14-May-2021
 * C source code generated on : Fri Mar 25 13:28:48 2022
 *
 * Target selection: bur_grt.tlc
 * Note: GRT includes extra infrastructure and instrumentation for prototyping
 * Embedded hardware selection: Intel->x86/Pentium
 * Code generation objectives: Unspecified
 * Validation result: Not run
 */

#ifndef RTWTYPES_H
#define RTWTYPES_H
#include "tmwtypes.h"
#ifndef POINTER_T
#define POINTER_T

typedef void * pointer_T;

#endif

/* Logical type definitions */
#if (!defined(__cplusplus))
#ifndef false
#define false                          (0U)
#endif

#ifndef true
#define true                           (1U)
#endif
#endif
#endif                                 /* RTWTYPES_H */
```

#### traj.c
```c
/********************************************************************
 * COPYRIGHT -- B&R Industrial Automation GmbH
 ********************************************************************
 * Program: traj_lib
 * File: traj_lib.c
 * Author: MartinV
 * Last modified by: MartinV
 * Created: 25-Mar-2022 13:28:52
 * Last modified: Fri Mar 25 13:28:41 2022
 * Model Version: 1.23
 * Description:
 * modified Comment:
 ********************************************************************
 * Implementation of program traj_lib
 ********************************************************************
 * Generated with B&R Automation Studio Target for Simulink V6.5
 * (GRT based)
 ********************************************************************/

#include <bur/plctypes.h>

#include "rtwtypes.h"
#include "rtmodel.h"

#define EXPAND_CONCAT(name1,name2) name1 ## name2
#define CONCAT(name1,name2) EXPAND_CONCAT(name1,name2)
#define RT_MODEL            CONCAT(MODEL,_rtModel)

#ifdef __cplusplus

extern "C" {

#endif

/* Defines */
#define SS_TERMINATE 4
#define SS_OUTPUT 3
#define SS_INITIALIZE 2

#ifdef __cplusplus

}

#endif

#ifdef __cplusplus
    unsigned long bur_heap_size = 6553500;
#endif

void traj(struct traj* inst)
{
  tag_RTM_generator_trajektorie_T* const generator_trajektorie_test_M = &(inst)->bur_generator_trajektorie_test;
	inst->bur_generator_trajektorie_test.blockIO = &(inst)->bur_B_generator_trajektorie_tes;

  switch (inst->ssMethodType)
  {
    case SS_INITIALIZE:

      /* call model initialize functions */
		/*memInit function */
		generator_trajektorie_test_initializeMemory(generator_trajektorie_test_M, inst);
		generator_trajektorie_test_initialize(generator_trajektorie_test_M, inst);
      break;

    case SS_OUTPUT:
      /* call model step functions */
		generator_trajektorie_test_step(generator_trajektorie_test_M, inst);
      break;

    case SS_TERMINATE:
      /* call model terminate function */
		generator_trajektorie_test_terminate(generator_trajektorie_test_M, inst);
	  break;
  }
}

/*****************************************************************************
   Function block sample time: 0.008
 *****************************************************************************/

/*****************************************************************************
   B&R Automation Studio Target for Simulink Version: V6.5.1 (03-Dec-2021)
 *****************************************************************************/
```

#### traj_lib.fun
```iecst
FUNCTION_BLOCK traj
	VAR_INPUT
		ssMethodType :  SINT;
		aktualny_uhol_x :  REAL :=  0; (**)
		aktualny_uhol_y :  REAL :=  0; (**)
		pozadovany_uhol_x :  REAL :=  0; (**)
		pozadovany_uhol_y :  REAL :=  0; (**)
		dlzka_pohybu :  REAL :=  0; (**)
	END_VAR
	VAR_OUTPUT
		trajektoria :  ARRAY[0..2,0..99] OF REAL :=  [300(0)]; (**)
		pocet_bodov_traj :  INT :=  0; (**)
	END_VAR
	VAR
		bur_B_generator_trajektorie_tes :  B_generator_trajektorie_test_T;
		bur_generator_trajektorie_test :  tag_RTM_generator_trajektorie_T;
	END_VAR
END_FUNCTION_BLOCK
```

### Library Logical/Library

#### Library.fun
```iecst
{REDUND_ERROR} FUNCTION_BLOCK suma (*TODO: Add your comment here*) (*$GROUP=User,$CAT=User,$GROUPICON=User.png,$CATICON=User.png*)
	VAR_INPUT
		a : BOOL;
		b : BOOL;
	END_VAR
	VAR_OUTPUT
		c : BOOL;
	END_VAR
END_FUNCTION_BLOCK

{REDUND_ERROR} FUNCTION_BLOCK transf_angle2dest (*TODO: Add your comment here*) (*$GROUP=User,$CAT=User,$GROUPICON=User.png,$CATICON=User.png*)
	VAR_INPUT
		AlfaX : LREAL;
		AlfaY : LREAL;
	END_VAR
	VAR_OUTPUT
		Dist_green : {REDUND_UNREPLICABLE} LREAL;
		Dist_yellow : {REDUND_UNREPLICABLE} LREAL;
		Dist_blue : {REDUND_UNREPLICABLE} LREAL;
		Test_value : LREAL;
	END_VAR
	VAR
		A1 : {REDUND_UNREPLICABLE} LREAL;
		A2 : {REDUND_UNREPLICABLE} LREAL;
		A3 : {REDUND_UNREPLICABLE} LREAL;
		B1 : {REDUND_UNREPLICABLE} LREAL;
		blue : {REDUND_UNREPLICABLE} ARRAY[0..3,0..0] OF LREAL;
		blue1 : {REDUND_UNREPLICABLE} ARRAY[0..3,0..0] OF LREAL;
		blue1_type : {REDUND_UNREPLICABLE} MTLinAlgMatrixType;
		blue_type : {REDUND_UNREPLICABLE} MTLinAlgMatrixType;
		Distance_blue : {REDUND_UNREPLICABLE} LREAL;
		Distance_green : {REDUND_UNREPLICABLE} LREAL;
		Distance_yellow : {REDUND_UNREPLICABLE} LREAL;
		green : {REDUND_UNREPLICABLE} ARRAY[0..3,0..0] OF LREAL;
		green1 : {REDUND_UNREPLICABLE} ARRAY[0..3,0..0] OF LREAL;
		green1_type : {REDUND_UNREPLICABLE} MTLinAlgMatrixType;
		green_type : {REDUND_UNREPLICABLE} MTLinAlgMatrixType;
		Htransform_base : {REDUND_UNREPLICABLE} ARRAY[0..3,0..3] OF LREAL;
		Htransform_base_type : {REDUND_UNREPLICABLE} MTLinAlgMatrixType;
		Htransform_yrelative : {REDUND_UNREPLICABLE} ARRAY[0..3,0..3] OF LREAL;
		Htransform_yrelative_type : {REDUND_UNREPLICABLE} MTLinAlgMatrixType;
		Rx01 : {REDUND_UNREPLICABLE} ARRAY[0..3,0..3] OF LREAL;
		Rx01_type : {REDUND_UNREPLICABLE} MTLinAlgMatrixType;
		Ry12 : {REDUND_UNREPLICABLE} ARRAY[0..3,0..3] OF LREAL;
		Ry12_type : {REDUND_UNREPLICABLE} MTLinAlgMatrixType;
		Tz23 : {REDUND_UNREPLICABLE} ARRAY[0..3,0..3] OF LREAL;
		Tz23_type : {REDUND_UNREPLICABLE} MTLinAlgMatrixType;
		Tz34 : {REDUND_UNREPLICABLE} ARRAY[0..3,0..3] OF LREAL;
		Tz34_type : {REDUND_UNREPLICABLE} MTLinAlgMatrixType;
		uholx_real_test : {REDUND_UNREPLICABLE} REAL;
		uholy_real_test : {REDUND_UNREPLICABLE} REAL;
		yellow : {REDUND_UNREPLICABLE} ARRAY[0..3,0..0] OF LREAL;
		yellow1 : {REDUND_UNREPLICABLE} ARRAY[0..3,0..0] OF LREAL;
		yellow1_type : {REDUND_UNREPLICABLE} MTLinAlgMatrixType;
		yellow_type : {REDUND_UNREPLICABLE} MTLinAlgMatrixType;
	END_VAR
END_FUNCTION_BLOCK

{REDUND_ERROR} {REDUND_UNREPLICABLE} FUNCTION_BLOCK Sin_signal (*TODO: Add your comment here*) (*$GROUP=User,$CAT=User,$GROUPICON=User.png,$CATICON=User.png*)
	VAR_INPUT
		time : {REDUND_UNREPLICABLE} REAL;
		Amplitude : {REDUND_UNREPLICABLE} REAL;
		frequency : {REDUND_UNREPLICABLE} REAL;
		phase : {REDUND_UNREPLICABLE} REAL;
	END_VAR
	VAR_OUTPUT
		angle : {REDUND_UNREPLICABLE} REAL;
	END_VAR
END_FUNCTION_BLOCK
```

#### suma.st
```iecst
(* TODO: Add your comment here *)
FUNCTION_BLOCK suma
	c:= a AND b;
END_FUNCTION_BLOCK
```

### Program Logical/Riadenie/Program (IEC)

#### Init.st
```iecst
PROGRAM _INIT
	(* Insert code here *)

END_PROGRAM
```

Listed in the project but not available here: Logical/Libraries/traj_lib/generator_trajektorie_test.h, Logical/Libraries/traj_lib/generator_trajektorie_test_private.h, Logical/Libraries/traj_lib/generator_trajektorie_test_types.h, Logical/Libraries/traj_lib/multiword_types.h, Logical/Libraries/traj_lib/rtGetInf.h, Logical/Libraries/traj_lib/rtGetNaN.c, Logical/Libraries/traj_lib/rt_defines.h, Logical/Libraries/traj_lib/rtmodel.h, Logical/Libraries/traj_lib/traj_lib.typ, Logical/Libraries/traj_lib/traj_lib.var, Logical/Libraries/traj_lib/rtw_continuous.h, Logical/Libraries/traj_lib/rtw_solver.h, Logical/Libraries/traj_lib/tmwtypes.h, Logical/Riadenie/riadenie.var
